KUKA KRL program: EPS_2_251626_SANMH03_A_20260107075954.src

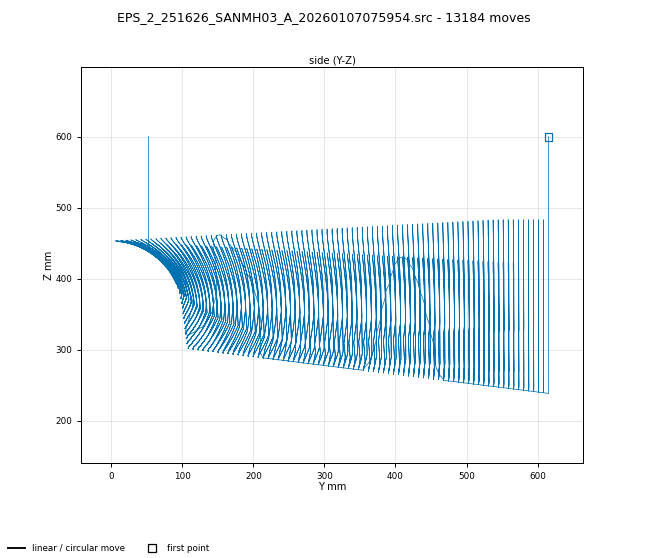
[picture p0: tool path of EPS_2_251626_SANMH03_A_20260107075954.src, 13184 of 13186 moves have a stored position in this frame; points joined in program order, loops and branches not executed]
&ACCESS RVP
&REL 4
&COMMENT QRS 19112012
&PARAM EDITMASK = *
DEF PART()
EXT BAS (BAS_COMMAND :IN,REAL :IN )
INT I
BAS (#INITMOV,0 )

;KUKA QRS Post kuka4.cps  Date:22-06-2017 !

File_ID=2961

QRS_PRE_INIT()

;Init var - Until changes are made in qrs_pre_init
Outlet_Square_prg=0
Inlet_1_Square_prg=0
Inlet_2_Square_prg=0
Inlet_3_Square_prg=0
Inlet_4_Square_prg=0
Inlet_5_Square_prg=0

Outlet_1={X 0.000, Y 541.230, Z 408.000, B 0.000, E1 0.000 }
Inlet_1={X 0.000, Y 545.490, Z 348.000, B 0.000, E1 180.000 }
Outlet_1_type=150
Inlet_1_type=150
;QRS#1=Sidecore dimensions
;QRS#2=150-6" PVC SDR 28
;QRS#3=150-6" PVC SDR 28
;QRS#4=
;QRS#5=
;QRS#6=
;QRS#7=
;QRS#8=
;QRS#9=10-06 PSX
;QRS#10=10-06 PSX
;QRS#11=
;QRS#12=
;QRS#13=
;QRS#14=
;QRS#15=
;QRS#16=1220x127x762 2,5'
;QRS#17=EPS Height
;QRS#18=483
;QRS#19=*
;QRS#20= UPDATED VERSION 22-06-2017
;QRS#21=*
Outlet_Square=070
Inlet_1_Square=070
Inlet_2_Square=0
Inlet_3_Square=0
Inlet_4_Square=0
Inlet_5_Square=0
Mill_Square=1
Outlet_Square_Prg=203
Inlet_1_Square_prg=203

QRS_INIT()

$ADVANCE=5

; T1
PTP {E1 173.651,E2 173.651}
PTP {X 0,Y 615.452,A -85,B 0,C 180,E1 173.651,E2 173.651,E3 0,E4 0,E5 0,E6 0}
QRS_SPEED_INIT()
LIN {X 0,Y 615.452,Z 600,A -85,B 0,C 180,E1 173.651,E2 173.651,E3 0,E4 0,E5 0,E6 0} C_VEL
LIN {X 0,Y 615.452,Z 248.689,A -85,B 0,C 180,E1 173.651,E2 173.651} C_VEL
LIN {X 0,Y 615.452,Z 240.511,A -85,B 0,C 180,E1 173.651,E2 173.651} C_VEL
LIN {X 0,Y 615.435,Z 238.511,A -85,B 0,C 180,E1 173.465,E2 173.465} C_VEL
LIN {X 0,Y 615.433,Z 238.511,A -85,B 0,C 180,E1 171.463,E2 171.463} C_VEL
LIN {X 0,Y 615.423,Z 238.51,A -85,B 0,C 180,E1 169.144,E2 169.144} C_VEL
LIN {X 0,Y 615.439,Z 238.509,A -85,B 0,C 180,E1 166.798,E2 166.798} C_VEL
LIN {X 0,Y 615.477,Z 238.513,A -85,B 0,C 180,E1 164.094,E2 164.094} C_VEL
LIN {X 0,Y 615.424,Z 238.51,A -85,B 0,C 180,E1 161.352,E2 161.352} C_VEL
LIN {X 0,Y 615.486,Z 238.507,A -85,B 0,C 180,E1 158.568,E2 158.568} C_VEL
LIN {X 0,Y 615.431,Z 238.51,A -85,B 0,C 180,E1 155.726,E2 155.726} C_VEL
LIN {X 0,Y 615.424,Z 238.51,A -85,B 0,C 180,E1 153.553,E2 153.553} C_VEL
LIN {X 0,Y 615.493,Z 238.51,A -85,B 0,C 180,E1 150.594,E2 150.594} C_VEL
LIN {X 0,Y 615.469,Z 238.512,A -85,B 0,C 180,E1 148.313,E2 148.313} C_VEL
LIN {X 0,Y 615.434,Z 238.51,A -85,B 0,C 180,E1 145.975,E2 145.975} C_VEL
LIN {X 0,Y 615.428,Z 238.509,A -85,B 0,C 180,E1 143.571,E2 143.571} C_VEL
LIN {X 0,Y 615.49,Z 238.506,A -85,B 0,C 180,E1 140.938,E2 140.938} C_VEL
LIN {X 0,Y 615.471,Z 238.512,A -85,B 0,C 180,E1 138.525,E2 138.525} C_VEL
LIN {X 0,Y 615.429,Z 238.509,A -85,B 0,C 180,E1 136.008,E2 136.008} C_VEL
LIN {X 0,Y 615.428,Z 238.509,A -85,B 0,C 180,E1 133.992,E2 133.992} C_VEL
LIN {X 0,Y 615.45,Z 238.507,A -85,B 0,C 180,E1 131.477,E2 131.477} C_VEL
LIN {X 0,Y 615.493,Z 238.513,A -85,B 0,C 180,E1 128.904,E2 128.904} C_VEL
LIN {X 0,Y 615.439,Z 238.51,A -85,B 0,C 180,E1 126.428,E2 126.428} C_VEL
LIN {X 0,Y 615.43,Z 238.508,A -85,B 0,C 180,E1 124.026,E2 124.026} C_VEL
LIN {X 0,Y 615.485,Z 238.516,A -85,B 0,C 180,E1 121.085,E2 121.085} C_VEL
LIN {X 0,Y 615.433,Z 238.509,A -85,B 0,C 180,E1 118.441,E2 118.441} C_VEL
LIN {X 0,Y 615.432,Z 238.509,A -85,B 0,C 180,E1 116.447,E2 116.447} C_VEL
LIN {X 0,Y 615.442,Z 238.507,A -85,B 0,C 180,E1 113.998,E2 113.998} C_VEL
LIN {X 0,Y 615.498,Z 238.508,A -85,B 0,C 180,E1 111.432,E2 111.432} C_VEL
LIN {X 0,Y 615.432,Z 238.509,A -85,B 0,C 180,E1 108.589,E2 108.589} C_VEL
LIN {X 0,Y 615.432,Z 238.508,A -85,B 0,C 180,E1 106.413,E2 106.413} C_VEL
LIN {X 0,Y 615.476,Z 238.722,A -85,B 0,C 180,E1 105.821,E2 105.821} C_VEL
LIN {X 0,Y 615.454,Z 250.521,A -85,B 0,C 180,E1 103.202,E2 103.202} C_VEL
LIN {X 0,Y 615.419,Z 261.215,A -85,B 0,C 180,E1 100.854,E2 100.854} C_VEL
LIN {X 0,Y 615.464,Z 264.873,A -85,B 0,C 180,E1 100.05,E2 100.05} C_VEL
LIN {X 0,Y 615.43,Z 339.723,A -85,B 0,C 180,E1 99.159,E2 99.159} C_VEL
LIN {X 0,Y 615.423,Z 347.907,A -85,B 0,C 180,E1 98.993,E2 98.993} C_VEL
LIN {X 0,Y 615.423,Z 356.463,A -85,B 0,C 180,E1 98.745,E2 98.745} C_VEL
LIN {X 0,Y 615.437,Z 364.07,A -85,B 0,C 180,E1 98.455,E2 98.455} C_VEL
LIN {X 0,Y 615.485,Z 372.58,A -85,B 0,C 180,E1 98.041,E2 98.041} C_VEL
LIN {X 0,Y 615.485,Z 380.745,A -85,B 0,C 180,E1 97.546,E2 97.546} C_VEL
LIN {X 0,Y 615.491,Z 387.386,A -85,B 0,C 180,E1 97.058,E2 97.058} C_VEL
LIN {X 0,Y 615.498,Z 393.181,A -85,B 0,C 180,E1 96.557,E2 96.557} C_VEL
LIN {X 0,Y 615.499,Z 399.532,A -85,B 0,C 180,E1 95.899,E2 95.899} C_VEL
LIN {X 0,Y 615.495,Z 405.982,A -85,B 0,C 180,E1 95.077,E2 95.077} C_VEL
LIN {X 0,Y 615.492,Z 411.121,A -85,B 0,C 180,E1 94.257,E2 94.257} C_VEL
LIN {X 0,Y 615.493,Z 415.885,A -85,B 0,C 180,E1 93.273,E2 93.273} C_VEL
LIN {X 0,Y 615.493,Z 418.199,A -85,B 0,C 180,E1 92.618,E2 92.618} C_VEL
LIN {X 0,Y 615.5,Z 419.975,A -85,B 0,C 180,E1 91.963,E2 91.963} C_VEL
LIN {X 0,Y 615.492,Z 421.266,A -85,B 0,C 180,E1 91.309,E2 91.309} C_VEL
LIN {X 0,Y 615.491,Z 422.083,A -85,B 0,C 180,E1 90.655,E2 90.655} C_VEL
LIN {X 0,Y 615.492,Z 422.384,A -85,B 0,C 180,E1 90,E2 90} C_VEL
LIN {X 0,Y 615.492,Z 422.125,A -85,B 0,C 180,E1 89.346,E2 89.346} C_VEL
LIN {X 0,Y 615.494,Z 421.394,A -85,B 0,C 180,E1 88.692,E2 88.692} C_VEL
LIN {X 0,Y 615.5,Z 420.195,A -85,B 0,C 180,E1 88.037,E2 88.037} C_VEL
LIN {X 0,Y 615.49,Z 417.377,A -85,B 0,C 180,E1 87.055,E2 87.055} C_VEL
LIN {X 0,Y 615.492,Z 414.811,A -85,B 0,C 180,E1 86.4,E2 86.4} C_VEL
LIN {X 0,Y 615.495,Z 409.745,A -85,B 0,C 180,E1 85.416,E2 85.416} C_VEL
LIN {X 0,Y 615.496,Z 404.29,A -85,B 0,C 180,E1 84.595,E2 84.595} C_VEL
LIN {X 0,Y 615.497,Z 397.456,A -85,B 0,C 180,E1 83.773,E2 83.773} C_VEL
LIN {X 0,Y 615.497,Z 390.421,A -85,B 0,C 180,E1 83.1,E2 83.1} C_VEL
LIN {X 0,Y 615.487,Z 382.077,A -85,B 0,C 180,E1 82.455,E2 82.455} C_VEL
LIN {X 0,Y 615.495,Z 374.202,A -85,B 0,C 180,E1 81.96,E2 81.96} C_VEL
LIN {X 0,Y 615.445,Z 366.093,A -85,B 0,C 180,E1 81.546,E2 81.546} C_VEL
LIN {X 0,Y 615.428,Z 357.89,A -85,B 0,C 180,E1 81.215,E2 81.215} C_VEL
LIN {X 0,Y 615.429,Z 349.874,A -85,B 0,C 180,E1 80.966,E2 80.966} C_VEL
LIN {X 0,Y 615.439,Z 340.208,A -85,B 0,C 180,E1 80.759,E2 80.759} C_VEL
LIN {X 0,Y 615.463,Z 264.814,A -85,B 0,C 180,E1 79.847,E2 79.847} C_VEL
LIN {X 0,Y 615.422,Z 253.988,A -85,B 0,C 180,E1 77.469,E2 77.469} C_VEL
LIN {X 0,Y 615.432,Z 243.324,A -85,B 0,C 180,E1 75.112,E2 75.112} C_VEL
LIN {X 0,Y 615.456,Z 238.508,A -85,B 0,C 180,E1 74.031,E2 74.031} C_VEL
LIN {X 0,Y 615.425,Z 238.51,A -85,B 0,C 180,E1 71.352,E2 71.352} C_VEL
LIN {X 0,Y 615.497,Z 238.511,A -85,B 0,C 180,E1 68.569,E2 68.569} C_VEL
LIN {X 0,Y 615.425,Z 238.509,A -85,B 0,C 180,E1 65.726,E2 65.726} C_VEL
LIN {X 0,Y 615.424,Z 238.51,A -85,B 0,C 180,E1 63.553,E2 63.553} C_VEL
LIN {X 0,Y 615.481,Z 238.51,A -85,B 0,C 180,E1 60.594,E2 60.594} C_VEL
LIN {X 0,Y 615.449,Z 238.508,A -85,B 0,C 180,E1 58.313,E2 58.313} C_VEL
LIN {X 0,Y 615.423,Z 238.51,A -85,B 0,C 180,E1 55.975,E2 55.975} C_VEL
LIN {X 0,Y 615.483,Z 238.512,A -85,B 0,C 180,E1 53.064,E2 53.064} C_VEL
LIN {X 0,Y 615.429,Z 238.51,A -85,B 0,C 180,E1 50.246,E2 50.246} C_VEL
LIN {X 0,Y 615.42,Z 238.511,A -85,B 0,C 180,E1 47.927,E2 47.927} C_VEL
LIN {X 0,Y 615.425,Z 238.511,A -85,B 0,C 180,E1 45.846,E2 45.846} C_VEL
LIN {X 0,Y 615.487,Z 238.512,A -85,B 0,C 180,E1 43.245,E2 43.245} C_VEL
LIN {X 0,Y 615.44,Z 238.509,A -85,B 0,C 180,E1 40.61,E2 40.61} C_VEL
LIN {X 0,Y 615.467,Z 238.509,A -85,B 0,C 180,E1 38.906,E2 38.906} C_VEL
LIN {X 0,Y 615.424,Z 238.51,A -85,B 0,C 180,E1 36.429,E2 36.429} C_VEL
LIN {X 0,Y 615.471,Z 238.513,A -85,B 0,C 180,E1 33.533,E2 33.533} C_VEL
LIN {X 0,Y 615.448,Z 238.509,A -85,B 0,C 180,E1 30.922,E2 30.922} C_VEL
LIN {X 0,Y 615.42,Z 238.51,A -85,B 0,C 180,E1 28.44,E2 28.44} C_VEL
LIN {X 0,Y 615.472,Z 238.512,A -85,B 0,C 180,E1 25.717,E2 25.717} C_VEL
LIN {X 0,Y 615.428,Z 238.51,A -85,B 0,C 180,E1 22.847,E2 22.847} C_VEL
LIN {X 0,Y 615.419,Z 238.511,A -85,B 0,C 180,E1 20.542,E2 20.542} C_VEL
LIN {X 0,Y 615.462,Z 238.512,A -85,B 0,C 180,E1 17.958,E2 17.958} C_VEL
LIN {X 0,Y 615.443,Z 238.51,A -85,B 0,C 180,E1 15.227,E2 15.227} C_VEL
LIN {X 0,Y 615.437,Z 238.51,A -85,B 0,C 180,E1 13.202,E2 13.202} C_VEL
LIN {X 0,Y 615.417,Z 238.511,A -85,B 0,C 180,E1 10.857,E2 10.857} C_VEL
LIN {X 0,Y 615.427,Z 238.511,A -85,B 0,C 180,E1 8.538,E2 8.538} C_VEL
LIN {X 0,Y 615.498,Z 238.511,A -85,B 0,C 180,E1 5.899,E2 5.899} C_VEL
LIN {X 0,Y 615.426,Z 238.511,A -85,B 0,C 180,E1 3.273,E2 3.273} C_VEL
LIN {X 0,Y 615.425,Z 238.511,A -85,B 0,C 180,E1 1.309,E2 1.309} C_VEL
LIN {X 0,Y 615.425,Z 238.511,A -85,B 0,C 180,E1 -0.654,E2 -0.654} C_VEL
LIN {X 0,Y 615.424,Z 238.511,A -85,B 0,C 180,E1 -2.618,E2 -2.618} C_VEL
LIN {X 0,Y 615.424,Z 238.511,A -85,B 0,C 180,E1 -4.585,E2 -4.585} C_VEL
LIN {X 0,Y 615.423,Z 238.511,A -85,B 0,C 180,E1 -6.557,E2 -6.557} C_VEL
LIN {X 0,Y 615.422,Z 238.511,A -85,B 0,C 180,E1 -8.537,E2 -8.537} C_VEL
LIN {X 0,Y 615.417,Z 238.512,A -85,B 0,C 180,E1 -10.857,E2 -10.857} C_VEL
LIN {X 0,Y 615.441,Z 238.512,A -85,B 0,C 180,E1 -13.202,E2 -13.202} C_VEL
LIN {X 0,Y 615.461,Z 238.511,A -85,B 0,C 180,E1 -15.906,E2 -15.906} C_VEL
LIN {X 0,Y 615.415,Z 238.512,A -85,B 0,C 180,E1 -18.648,E2 -18.648} C_VEL
LIN {X 0,Y 615.493,Z 238.512,A -85,B 0,C 180,E1 -21.432,E2 -21.432} C_VEL
LIN {X 0,Y 615.417,Z 238.511,A -85,B 0,C 180,E1 -24.275,E2 -24.275} C_VEL
LIN {X 0,Y 615.415,Z 238.512,A -85,B 0,C 180,E1 -26.447,E2 -26.447} C_VEL
LIN {X 0,Y 615.478,Z 238.514,A -85,B 0,C 180,E1 -29.407,E2 -29.407} C_VEL
LIN {X 0,Y 615.445,Z 238.511,A -85,B 0,C 180,E1 -31.688,E2 -31.688} C_VEL
LIN {X 0,Y 615.418,Z 238.512,A -85,B 0,C 180,E1 -34.026,E2 -34.026} C_VEL
LIN {X 0,Y 615.464,Z 238.513,A -85,B 0,C 180,E1 -36.935,E2 -36.935} C_VEL
LIN {X 0,Y 615.422,Z 238.512,A -85,B 0,C 180,E1 -39.755,E2 -39.755} C_VEL
LIN {X 0,Y 615.413,Z 238.512,A -85,B 0,C 180,E1 -42.073,E2 -42.073} C_VEL
LIN {X 0,Y 615.415,Z 238.512,A -85,B 0,C 180,E1 -44.156,E2 -44.156} C_VEL
LIN {X 0,Y 615.471,Z 238.512,A -85,B 0,C 180,E1 -46.755,E2 -46.755} C_VEL
LIN {X 0,Y 615.435,Z 238.512,A -85,B 0,C 180,E1 -49.39,E2 -49.39} C_VEL
LIN {X 0,Y 615.465,Z 238.512,A -85,B 0,C 180,E1 -51.095,E2 -51.095} C_VEL
LIN {X 0,Y 615.417,Z 238.512,A -85,B 0,C 180,E1 -53.571,E2 -53.571} C_VEL
LIN {X 0,Y 615.46,Z 238.512,A -85,B 0,C 180,E1 -56.47,E2 -56.47} C_VEL
LIN {X 0,Y 615.444,Z 238.512,A -85,B 0,C 180,E1 -59.078,E2 -59.078} C_VEL
LIN {X 0,Y 615.412,Z 238.512,A -85,B 0,C 180,E1 -61.563,E2 -61.563} C_VEL
LIN {X 0,Y 615.409,Z 238.513,A -85,B 0,C 180,E1 -63.553,E2 -63.553} C_VEL
LIN {X 0,Y 615.431,Z 238.512,A -85,B 0,C 180,E1 -66.003,E2 -66.003} C_VEL
LIN {X 0,Y 615.422,Z 238.609,A -85,B 0,C 180,E1 -67.838,E2 -67.838} C_VEL
LIN {X 0,Y 615.475,Z 257.737,A -85,B 0,C 180,E1 -70.662,E2 -70.662} C_VEL
LIN {X 0,Y 615.482,Z 276.679,A -85,B 0,C 180,E1 -73.414,E2 -73.414} C_VEL
LIN {X 0,Y 615.488,Z 296.786,A -85,B 0,C 180,E1 -76.295,E2 -76.295} C_VEL
LIN {X 0,Y 615.448,Z 316.82,A -85,B 0,C 180,E1 -79.131,E2 -79.131} C_VEL
LIN {X 0,Y 615.46,Z 322.04,A -85,B 0,C 180,E1 -79.868,E2 -79.868} C_VEL
LIN {X 0,Y 615.446,Z 399.981,A -85,B 0,C 180,E1 -80.801,E2 -80.801} C_VEL
LIN {X 0,Y 615.436,Z 409.728,A -85,B 0,C 180,E1 -81.008,E2 -81.008} C_VEL
LIN {X 0,Y 615.436,Z 420.18,A -85,B 0,C 180,E1 -81.339,E2 -81.339} C_VEL
LIN {X 0,Y 615.471,Z 430.44,A -85,B 0,C 180,E1 -81.794,E2 -81.794} C_VEL
LIN {X 0,Y 615.489,Z 440.204,A -85,B 0,C 180,E1 -82.372,E2 -82.372} C_VEL
LIN {X 0,Y 615.494,Z 447.938,A -85,B 0,C 180,E1 -82.942,E2 -82.942} C_VEL
LIN {X 0,Y 615.497,Z 455.338,A -85,B 0,C 180,E1 -83.608,E2 -83.608} C_VEL
LIN {X 0,Y 615.498,Z 462.74,A -85,B 0,C 180,E1 -84.431,E2 -84.431} C_VEL
LIN {X 0,Y 615.497,Z 468.535,A -85,B 0,C 180,E1 -85.252,E2 -85.252} C_VEL
LIN {X 0,Y 615.496,Z 473.102,A -85,B 0,C 180,E1 -86.072,E2 -86.072} C_VEL
LIN {X 0,Y 615.492,Z 476.07,A -85,B 0,C 180,E1 -86.727,E2 -86.727} C_VEL
LIN {X 0,Y 615.494,Z 478.358,A -85,B 0,C 180,E1 -87.383,E2 -87.383} C_VEL
LIN {X 0,Y 615.5,Z 480.086,A -85,B 0,C 180,E1 -88.037,E2 -88.037} C_VEL
LIN {X 0,Y 615.493,Z 481.33,A -85,B 0,C 180,E1 -88.692,E2 -88.692} C_VEL
LIN {X 0,Y 615.492,Z 482.104,A -85,B 0,C 180,E1 -89.346,E2 -89.346} C_VEL
LIN {X 0,Y 615.491,Z 482.389,A -85,B 0,C 180,E1 -90,E2 -90} C_VEL
LIN {X 0,Y 615.491,Z 482.104,A -85,B 0,C 180,E1 -90.655,E2 -90.655} C_VEL
LIN {X 0,Y 615.493,Z 481.329,A -85,B 0,C 180,E1 -91.309,E2 -91.309} C_VEL
LIN {X 0,Y 615.5,Z 480.084,A -85,B 0,C 180,E1 -91.963,E2 -91.963} C_VEL
LIN {X 0,Y 615.488,Z 477.22,A -85,B 0,C 180,E1 -92.946,E2 -92.946} C_VEL
LIN {X 0,Y 615.491,Z 474.602,A -85,B 0,C 180,E1 -93.601,E2 -93.601} C_VEL
LIN {X 0,Y 615.495,Z 469.48,A -85,B 0,C 180,E1 -94.585,E2 -94.585} C_VEL
LIN {X 0,Y 615.495,Z 463.966,A -85,B 0,C 180,E1 -95.406,E2 -95.406} C_VEL
LIN {X 0,Y 615.498,Z 457.015,A -85,B 0,C 180,E1 -96.228,E2 -96.228} C_VEL
LIN {X 0,Y 615.496,Z 449.857,A -85,B 0,C 180,E1 -96.901,E2 -96.901} C_VEL
LIN {X 0,Y 615.485,Z 442.618,A -85,B 0,C 180,E1 -97.463,E2 -97.463} C_VEL
LIN {X 0,Y 615.495,Z 434.863,A -85,B 0,C 180,E1 -97.958,E2 -97.958} C_VEL
LIN {X 0,Y 615.454,Z 426.917,A -85,B 0,C 180,E1 -98.372,E2 -98.372} C_VEL
LIN {X 0,Y 615.434,Z 417.763,A -85,B 0,C 180,E1 -98.744,E2 -98.744} C_VEL
LIN {X 0,Y 615.436,Z 409.701,A -85,B 0,C 180,E1 -98.993,E2 -98.993} C_VEL
LIN {X 0,Y 615.446,Z 399.938,A -85,B 0,C 180,E1 -99.2,E2 -99.2} C_VEL
LIN {X 0,Y 615.46,Z 322.035,A -85,B 0,C 180,E1 -100.133,E2 -100.133} C_VEL
LIN {X 0,Y 615.468,Z 303.881,A -85,B 0,C 180,E1 -102.698,E2 -102.698} C_VEL
LIN {X 0,Y 615.486,Z 283.774,A -85,B 0,C 180,E1 -105.566,E2 -105.566} C_VEL
LIN {X 0,Y 615.469,Z 263.911,A -85,B 0,C 180,E1 -108.437,E2 -108.437} C_VEL
LIN {X 0,Y 615.439,Z 247.065,A -85,B 0,C 180,E1 -110.908,E2 -110.908} C_VEL
LIN {X 0,Y 615.42,Z 238.512,A -85,B 0,C 180,E1 -112.187,E2 -112.187} C_VEL
LIN {X 0,Y 615.414,Z 238.512,A -85,B 0,C 180,E1 -114.275,E2 -114.275} C_VEL
LIN {X 0,Y 615.41,Z 238.513,A -85,B 0,C 180,E1 -116.448,E2 -116.448} C_VEL
LIN {X 0,Y 615.478,Z 238.516,A -85,B 0,C 180,E1 -119.407,E2 -119.407} C_VEL
LIN {X 0,Y 615.446,Z 238.512,A -85,B 0,C 180,E1 -121.688,E2 -121.688} C_VEL
LIN {X 0,Y 615.417,Z 238.512,A -85,B 0,C 180,E1 -124.027,E2 -124.027} C_VEL
LIN {X 0,Y 615.463,Z 238.512,A -85,B 0,C 180,E1 -126.934,E2 -126.934} C_VEL
LIN {X 0,Y 615.426,Z 238.512,A -85,B 0,C 180,E1 -129.755,E2 -129.755} C_VEL
LIN {X 0,Y 615.414,Z 238.512,A -85,B 0,C 180,E1 -132.073,E2 -132.073} C_VEL
LIN {X 0,Y 615.415,Z 238.512,A -85,B 0,C 180,E1 -134.156,E2 -134.156} C_VEL
LIN {X 0,Y 615.414,Z 238.512,A -85,B 0,C 180,E1 -136.01,E2 -136.01} C_VEL
LIN {X 0,Y 615.445,Z 238.511,A -85,B 0,C 180,E1 -138.523,E2 -138.523} C_VEL
LIN {X 0,Y 615.472,Z 238.512,A -85,B 0,C 180,E1 -141.095,E2 -141.095} C_VEL
LIN {X 0,Y 615.422,Z 238.512,A -85,B 0,C 180,E1 -143.571,E2 -143.571} C_VEL
LIN {X 0,Y 615.418,Z 238.511,A -85,B 0,C 180,E1 -145.974,E2 -145.974} C_VEL
LIN {X 0,Y 615.443,Z 238.511,A -85,B 0,C 180,E1 -148.312,E2 -148.312} C_VEL
LIN {X 0,Y 615.478,Z 238.513,A -85,B 0,C 180,E1 -150.593,E2 -150.593} C_VEL
LIN {X 0,Y 615.418,Z 238.511,A -85,B 0,C 180,E1 -153.553,E2 -153.553} C_VEL
LIN {X 0,Y 615.433,Z 238.511,A -85,B 0,C 180,E1 -156.003,E2 -156.003} C_VEL
LIN {X 0,Y 615.498,Z 238.513,A -85,B 0,C 180,E1 -158.569,E2 -158.569} C_VEL
LIN {X 0,Y 615.418,Z 238.511,A -85,B 0,C 180,E1 -161.415,E2 -161.415} C_VEL
LIN {X 0,Y 615.462,Z 238.51,A -85,B 0,C 180,E1 -164.094,E2 -164.094} C_VEL
LIN {X 0,Y 615.445,Z 238.512,A -85,B 0,C 180,E1 -166.798,E2 -166.798} C_VEL
LIN {X 0,Y 615.421,Z 238.511,A -85,B 0,C 180,E1 -169.144,E2 -169.144} C_VEL
LIN {X 0,Y 615.424,Z 238.51,A -85,B 0,C 180,E1 -171.463,E2 -171.463} C_VEL
LIN {X 0,Y 615.496,Z 238.508,A -85,B 0,C 180,E1 -174.102,E2 -174.102} C_VEL
LIN {X 0,Y 615.435,Z 238.511,A -85,B 0,C 180,E1 -176.727,E2 -176.727} C_VEL
LIN {X 0,Y 615.435,Z 238.511,A -85,B 0,C 180,E1 -178.691,E2 -178.691} C_VEL
LIN {X 0,Y 615.434,Z 238.511,A -85,B 0,C 180,E1 -180.654,E2 -180.654} C_VEL
LIN {X 0,Y 615.435,Z 238.511,A -85,B 0,C 180,E1 -182.618,E2 -182.618} C_VEL
LIN {X 0,Y 615.434,Z 238.511,A -85,B 0,C 180,E1 -184.585,E2 -184.585} C_VEL
LIN {X 0,Y 615.435,Z 238.511,A -85,B 0,C 180,E1 -186.535,E2 -186.535} C_VEL
LIN {X 0,Y 614.753,Z 238.655,A -85,B 0,C 180,E1 -187.081,E2 -187.081} C_VEL
LIN {X 0,Y 611.913,Z 239.08,A -85,B 0,C 180,E1 -187.967,E2 -187.967} C_VEL
LIN {X 0,Y 609.529,Z 239.382,A -85,B 0,C 180,E1 -188.68,E2 -188.68} C_VEL
LIN {X 0,Y 608.51,Z 239.496,A -85,B 0,C 180,E1 -189.23,E2 -189.23} C_VEL
LIN {X 0,Y 608.429,Z 239.505,A -85,B 0,C 180,E1 -189.416,E2 -189.416} C_VEL
LIN {X 0,Y 608.449,Z 239.509,A -85,B 0,C 180,E1 -192,E2 -192} C_VEL
LIN {X 0,Y 608.396,Z 239.507,A -85,B 0,C 180,E1 -194.723,E2 -194.723} C_VEL
LIN {X 0,Y 608.428,Z 239.509,A -85,B 0,C 180,E1 -197.477,E2 -197.477} C_VEL
LIN {X 0,Y 608.42,Z 239.506,A -85,B 0,C 180,E1 -200.276,E2 -200.276} C_VEL
LIN {X 0,Y 608.397,Z 239.507,A -85,B 0,C 180,E1 -202.462,E2 -202.462} C_VEL
LIN {X 0,Y 608.412,Z 239.505,A -85,B 0,C 180,E1 -204.573,E2 -204.573} C_VEL
LIN {X 0,Y 608.46,Z 239.504,A -85,B 0,C 180,E1 -207.204,E2 -207.204} C_VEL
LIN {X 0,Y 608.419,Z 239.507,A -85,B 0,C 180,E1 -209.963,E2 -209.963} C_VEL
LIN {X 0,Y 608.412,Z 239.505,A -85,B 0,C 180,E1 -212.515,E2 -212.515} C_VEL
LIN {X 0,Y 608.417,Z 239.507,A -85,B 0,C 180,E1 -214.901,E2 -214.901} C_VEL
LIN {X 0,Y 608.438,Z 239.506,A -85,B 0,C 180,E1 -217.749,E2 -217.749} C_VEL
LIN {X 0,Y 608.403,Z 239.506,A -85,B 0,C 180,E1 -220.323,E2 -220.323} C_VEL
LIN {X 0,Y 608.447,Z 239.507,A -85,B 0,C 180,E1 -222.96,E2 -222.96} C_VEL
LIN {X 0,Y 608.414,Z 239.507,A -85,B 0,C 180,E1 -225.74,E2 -225.74} C_VEL
LIN {X 0,Y 608.413,Z 239.505,A -85,B 0,C 180,E1 -227.934,E2 -227.934} C_VEL
LIN {X 0,Y 608.438,Z 239.506,A -85,B 0,C 180,E1 -230.706,E2 -230.706} C_VEL
LIN {X 0,Y 608.454,Z 239.51,A -85,B 0,C 180,E1 -233.085,E2 -233.085} C_VEL
LIN {X 0,Y 608.437,Z 239.504,A -85,B 0,C 180,E1 -235.528,E2 -235.528} C_VEL
LIN {X 0,Y 608.422,Z 239.504,A -85,B 0,C 180,E1 -237.903,E2 -237.903} C_VEL
LIN {X 0,Y 608.433,Z 239.504,A -85,B 0,C 180,E1 -240.218,E2 -240.218} C_VEL
LIN {X 0,Y 608.48,Z 239.507,A -85,B 0,C 180,E1 -242.793,E2 -242.793} C_VEL
LIN {X 0,Y 608.421,Z 239.505,A -85,B 0,C 180,E1 -245.427,E2 -245.427} C_VEL
LIN {X 0,Y 608.458,Z 239.503,A -85,B 0,C 180,E1 -248.308,E2 -248.308} C_VEL
LIN {X 0,Y 608.418,Z 239.506,A -85,B 0,C 180,E1 -251.299,E2 -251.299} C_VEL
LIN {X 0,Y 608.455,Z 239.58,A -85,B 0,C 180,E1 -254.142,E2 -254.142} C_VEL
LIN {X 0,Y 608.411,Z 252.299,A -85,B 0,C 180,E1 -256.982,E2 -256.982} C_VEL
LIN {X 0,Y 608.401,Z 264.922,A -85,B 0,C 180,E1 -259.769,E2 -259.769} C_VEL
LIN {X 0,Y 608.426,Z 265.209,A -85,B 0,C 180,E1 -259.833,E2 -259.833} C_VEL
LIN {X 0,Y 608.458,Z 340.233,A -85,B 0,C 180,E1 -260.736,E2 -260.736} C_VEL
LIN {X 0,Y 608.448,Z 349.939,A -85,B 0,C 180,E1 -260.945,E2 -260.945} C_VEL
LIN {X 0,Y 608.433,Z 361.53,A -85,B 0,C 180,E1 -261.321,E2 -261.321} C_VEL
LIN {X 0,Y 608.462,Z 371.427,A -85,B 0,C 180,E1 -261.782,E2 -261.782} C_VEL
LIN {X 0,Y 608.468,Z 379.881,A -85,B 0,C 180,E1 -262.283,E2 -262.283} C_VEL
LIN {X 0,Y 608.459,Z 387.85,A -85,B 0,C 180,E1 -262.867,E2 -262.867} C_VEL
LIN {X 0,Y 608.468,Z 394.901,A -85,B 0,C 180,E1 -263.496,E2 -263.496} C_VEL
LIN {X 0,Y 608.458,Z 401.393,A -85,B 0,C 180,E1 -264.199,E2 -264.199} C_VEL
LIN {X 0,Y 608.437,Z 407.639,A -85,B 0,C 180,E1 -265.03,E2 -265.03} C_VEL
LIN {X 0,Y 608.434,Z 413.423,A -85,B 0,C 180,E1 -266.026,E2 -266.026} C_VEL
LIN {X 0,Y 608.447,Z 417.629,A -85,B 0,C 180,E1 -267.02,E2 -267.02} C_VEL
LIN {X 0,Y 608.444,Z 420.569,A -85,B 0,C 180,E1 -268.014,E2 -268.014} C_VEL
LIN {X 0,Y 608.445,Z 421.869,A -85,B 0,C 180,E1 -268.676,E2 -268.676} C_VEL
LIN {X 0,Y 608.434,Z 422.692,A -85,B 0,C 180,E1 -269.338,E2 -269.338} C_VEL
LIN {X 0,Y 608.432,Z 422.995,A -85,B 0,C 180,E1 -270,E2 -270} C_VEL
LIN {X 0,Y 608.435,Z 422.735,A -85,B 0,C 180,E1 -270.661,E2 -270.661} C_VEL
LIN {X 0,Y 608.446,Z 421.998,A -85,B 0,C 180,E1 -271.323,E2 -271.323} C_VEL
LIN {X 0,Y 608.444,Z 420.788,A -85,B 0,C 180,E1 -271.985,E2 -271.985} C_VEL
LIN {X 0,Y 608.445,Z 417.943,A -85,B 0,C 180,E1 -272.979,E2 -272.979} C_VEL
LIN {X 0,Y 608.446,Z 415.353,A -85,B 0,C 180,E1 -273.642,E2 -273.642} C_VEL
LIN {X 0,Y 608.445,Z 410.247,A -85,B 0,C 180,E1 -274.637,E2 -274.637} C_VEL
LIN {X 0,Y 608.461,Z 404.751,A -85,B 0,C 180,E1 -275.468,E2 -275.468} C_VEL
LIN {X 0,Y 608.454,Z 397.149,A -85,B 0,C 180,E1 -276.374,E2 -276.374} C_VEL
LIN {X 0,Y 608.463,Z 388.952,A -85,B 0,C 180,E1 -277.132,E2 -277.132} C_VEL
LIN {X 0,Y 608.469,Z 381.204,A -85,B 0,C 180,E1 -277.716,E2 -277.716} C_VEL
LIN {X 0,Y 608.47,Z 373.04,A -85,B 0,C 180,E1 -278.217,E2 -278.217} C_VEL
LIN {X 0,Y 608.434,Z 364.54,A -85,B 0,C 180,E1 -278.636,E2 -278.636} C_VEL
LIN {X 0,Y 608.422,Z 353.345,A -85,B 0,C 180,E1 -279.055,E2 -279.055} C_VEL
LIN {X 0,Y 608.461,Z 341.959,A -85,B 0,C 180,E1 -279.327,E2 -279.327} C_VEL
LIN {X 0,Y 608.469,Z 321.042,A -85,B 0,C 180,E1 -279.599,E2 -279.599} C_VEL
LIN {X 0,Y 608.41,Z 265.143,A -85,B 0,C 180,E1 -280.272,E2 -280.272} C_VEL
LIN {X 0,Y 608.402,Z 252.707,A -85,B 0,C 180,E1 -283.017,E2 -283.017} C_VEL
LIN {X 0,Y 608.449,Z 240.462,A -85,B 0,C 180,E1 -285.75,E2 -285.75} C_VEL
LIN {X 0,Y 608.44,Z 239.504,A -85,B 0,C 180,E1 -286.008,E2 -286.008} C_VEL
LIN {X 0,Y 608.43,Z 239.505,A -85,B 0,C 180,E1 -288.87,E2 -288.87} C_VEL
LIN {X 0,Y 608.456,Z 239.505,A -85,B 0,C 180,E1 -291.692,E2 -291.692} C_VEL
LIN {X 0,Y 608.414,Z 239.506,A -85,B 0,C 180,E1 -294.572,E2 -294.572} C_VEL
LIN {X 0,Y 608.471,Z 239.508,A -85,B 0,C 180,E1 -297.206,E2 -297.206} C_VEL
LIN {X 0,Y 608.406,Z 239.506,A -85,B 0,C 180,E1 -299.961,E2 -299.961} C_VEL
LIN {X 0,Y 608.413,Z 239.506,A -85,B 0,C 180,E1 -302.515,E2 -302.515} C_VEL
LIN {X 0,Y 608.421,Z 239.511,A -85,B 0,C 180,E1 -304.901,E2 -304.901} C_VEL
LIN {X 0,Y 608.429,Z 239.504,A -85,B 0,C 180,E1 -307.749,E2 -307.749} C_VEL
LIN {X 0,Y 608.398,Z 239.508,A -85,B 0,C 180,E1 -310.323,E2 -310.323} C_VEL
LIN {X 0,Y 608.447,Z 239.511,A -85,B 0,C 180,E1 -312.96,E2 -312.96} C_VEL
LIN {X 0,Y 608.404,Z 239.506,A -85,B 0,C 180,E1 -315.74,E2 -315.74} C_VEL
LIN {X 0,Y 608.406,Z 239.506,A -85,B 0,C 180,E1 -317.934,E2 -317.934} C_VEL
LIN {X 0,Y 608.434,Z 239.512,A -85,B 0,C 180,E1 -320.706,E2 -320.706} C_VEL
LIN {X 0,Y 608.433,Z 239.507,A -85,B 0,C 180,E1 -323.083,E2 -323.083} C_VEL
LIN {X 0,Y 608.42,Z 239.504,A -85,B 0,C 180,E1 -325.527,E2 -325.527} C_VEL
LIN {X 0,Y 608.418,Z 239.505,A -85,B 0,C 180,E1 -327.903,E2 -327.903} C_VEL
LIN {X 0,Y 608.438,Z 239.507,A -85,B 0,C 180,E1 -330.219,E2 -330.219} C_VEL
LIN {X 0,Y 608.398,Z 239.508,A -85,B 0,C 180,E1 -333.223,E2 -333.223} C_VEL
LIN {X 0,Y 608.407,Z 239.506,A -85,B 0,C 180,E1 -335.427,E2 -335.427} C_VEL
LIN {X 0,Y 608.45,Z 239.51,A -85,B 0,C 180,E1 -338.308,E2 -338.308} C_VEL
LIN {X 0,Y 608.406,Z 239.506,A -85,B 0,C 180,E1 -341.3,E2 -341.3} C_VEL
LIN {X 0,Y 608.428,Z 239.508,A -85,B 0,C 180,E1 -343.905,E2 -343.905} C_VEL
LIN {X 0,Y 608.428,Z 239.507,A -85,B 0,C 180,E1 -346.643,E2 -346.643} C_VEL
LIN {X 0,Y 608.402,Z 239.507,A -85,B 0,C 180,E1 -349.349,E2 -349.349} C_VEL
LIN {X 0,Y 608.465,Z 239.508,A -85,B 0,C 180,E1 -352.033,E2 -352.033} C_VEL
LIN {X 0,Y 608.413,Z 239.506,A -85,B 0,C 180,E1 -354.698,E2 -354.698} C_VEL
LIN {X 0,Y 608.424,Z 239.505,A -85,B 0,C 180,E1 -357.352,E2 -357.352} C_VEL
LIN {X 0,Y 608.47,Z 239.507,A -85,B 0,C 180,E1 -360,E2 -360} C_VEL
LIN {X 0,Y 608.42,Z 239.505,A -85,B 0,C 180,E1 -362.648,E2 -362.648} C_VEL
LIN {X 0,Y 608.419,Z 239.507,A -85,B 0,C 180,E1 -365.302,E2 -365.302} C_VEL
LIN {X 0,Y 608.463,Z 239.506,A -85,B 0,C 180,E1 -367.967,E2 -367.967} C_VEL
LIN {X 0,Y 608.4,Z 239.507,A -85,B 0,C 180,E1 -370.651,E2 -370.651} C_VEL
LIN {X 0,Y 608.428,Z 239.509,A -85,B 0,C 180,E1 -373.357,E2 -373.357} C_VEL
LIN {X 0,Y 608.422,Z 239.507,A -85,B 0,C 180,E1 -376.095,E2 -376.095} C_VEL
LIN {X 0,Y 608.422,Z 239.505,A -85,B 0,C 180,E1 -378.871,E2 -378.871} C_VEL
LIN {X 0,Y 608.451,Z 239.507,A -85,B 0,C 180,E1 -381.692,E2 -381.692} C_VEL
LIN {X 0,Y 608.404,Z 239.506,A -85,B 0,C 180,E1 -384.573,E2 -384.573} C_VEL
LIN {X 0,Y 608.459,Z 239.507,A -85,B 0,C 180,E1 -387.205,E2 -387.205} C_VEL
LIN {X 0,Y 608.401,Z 239.508,A -85,B 0,C 180,E1 -389.962,E2 -389.962} C_VEL
LIN {X 0,Y 608.404,Z 239.507,A -85,B 0,C 180,E1 -392.515,E2 -392.515} C_VEL
LIN {X 0,Y 608.412,Z 239.511,A -85,B 0,C 180,E1 -394.901,E2 -394.901} C_VEL
LIN {X 0,Y 608.423,Z 239.505,A -85,B 0,C 180,E1 -397.75,E2 -397.75} C_VEL
LIN {X 0,Y 608.396,Z 239.508,A -85,B 0,C 180,E1 -400.324,E2 -400.324} C_VEL
LIN {X 0,Y 608.437,Z 239.512,A -85,B 0,C 180,E1 -402.961,E2 -402.961} C_VEL
LIN {X 0,Y 608.398,Z 239.507,A -85,B 0,C 180,E1 -405.742,E2 -405.742} C_VEL
LIN {X 0,Y 608.398,Z 239.507,A -85,B 0,C 180,E1 -407.934,E2 -407.934} C_VEL
LIN {X 0,Y 608.43,Z 239.511,A -85,B 0,C 180,E1 -410.707,E2 -410.707} C_VEL
LIN {X 0,Y 608.431,Z 239.508,A -85,B 0,C 180,E1 -413.084,E2 -413.084} C_VEL
LIN {X 0,Y 608.416,Z 239.505,A -85,B 0,C 180,E1 -415.528,E2 -415.528} C_VEL
LIN {X 0,Y 608.409,Z 239.506,A -85,B 0,C 180,E1 -417.903,E2 -417.903} C_VEL
LIN {X 0,Y 608.425,Z 239.507,A -85,B 0,C 180,E1 -420.219,E2 -420.219} C_VEL
LIN {X 0,Y 608.456,Z 239.507,A -85,B 0,C 180,E1 -422.797,E2 -422.797} C_VEL
LIN {X 0,Y 608.401,Z 239.507,A -85,B 0,C 180,E1 -425.427,E2 -425.427} C_VEL
LIN {X 0,Y 608.423,Z 239.662,A -85,B 0,C 180,E1 -427.727,E2 -427.727} C_VEL
LIN {X 0,Y 608.49,Z 251.996,A -85,B 0,C 180,E1 -429.576,E2 -429.576} C_VEL
LIN {X 0,Y 608.507,Z 270.816,A -85,B 0,C 180,E1 -432.352,E2 -432.352} C_VEL
LIN {X 0,Y 608.482,Z 289.806,A -85,B 0,C 180,E1 -435.109,E2 -435.109} C_VEL
LIN {X 0,Y 608.453,Z 308.795,A -85,B 0,C 180,E1 -437.831,E2 -437.831} C_VEL
LIN {X 0,Y 608.436,Z 322.296,A -85,B 0,C 180,E1 -439.75,E2 -439.75} C_VEL
LIN {X 0,Y 608.473,Z 400.467,A -85,B 0,C 180,E1 -440.695,E2 -440.695} C_VEL
LIN {X 0,Y 608.437,Z 410.09,A -85,B 0,C 180,E1 -440.904,E2 -440.904} C_VEL
LIN {X 0,Y 608.426,Z 421.627,A -85,B 0,C 180,E1 -441.28,E2 -441.28} C_VEL
LIN {X 0,Y 608.47,Z 432.239,A -85,B 0,C 180,E1 -441.783,E2 -441.783} C_VEL
LIN {X 0,Y 608.468,Z 440.547,A -85,B 0,C 180,E1 -442.284,E2 -442.284} C_VEL
LIN {X 0,Y 608.46,Z 448.405,A -85,B 0,C 180,E1 -442.868,E2 -442.868} C_VEL
LIN {X 0,Y 608.466,Z 455.359,A -85,B 0,C 180,E1 -443.496,E2 -443.496} C_VEL
LIN {X 0,Y 608.47,Z 463.194,A -85,B 0,C 180,E1 -444.366,E2 -444.366} C_VEL
LIN {X 0,Y 608.448,Z 469.029,A -85,B 0,C 180,E1 -445.197,E2 -445.197} C_VEL
LIN {X 0,Y 608.434,Z 473.632,A -85,B 0,C 180,E1 -446.026,E2 -446.026} C_VEL
LIN {X 0,Y 608.424,Z 476.623,A -85,B 0,C 180,E1 -446.689,E2 -446.689} C_VEL
LIN {X 0,Y 608.423,Z 478.932,A -85,B 0,C 180,E1 -447.352,E2 -447.352} C_VEL
LIN {X 0,Y 608.444,Z 480.679,A -85,B 0,C 180,E1 -448.015,E2 -448.015} C_VEL
LIN {X 0,Y 608.445,Z 481.934,A -85,B 0,C 180,E1 -448.677,E2 -448.677} C_VEL
LIN {X 0,Y 608.434,Z 482.714,A -85,B 0,C 180,E1 -449.339,E2 -449.339} C_VEL
LIN {X 0,Y 608.431,Z 483,A -85,B 0,C 180,E1 -450,E2 -450} C_VEL
LIN {X 0,Y 608.434,Z 482.713,A -85,B 0,C 180,E1 -450.662,E2 -450.662} C_VEL
LIN {X 0,Y 608.446,Z 481.933,A -85,B 0,C 180,E1 -451.324,E2 -451.324} C_VEL
LIN {X 0,Y 608.444,Z 480.677,A -85,B 0,C 180,E1 -451.986,E2 -451.986} C_VEL
LIN {X 0,Y 608.444,Z 477.785,A -85,B 0,C 180,E1 -452.98,E2 -452.98} C_VEL
LIN {X 0,Y 608.445,Z 475.145,A -85,B 0,C 180,E1 -453.643,E2 -453.643} C_VEL
LIN {X 0,Y 608.431,Z 469.983,A -85,B 0,C 180,E1 -454.638,E2 -454.638} C_VEL
LIN {X 0,Y 608.46,Z 464.427,A -85,B 0,C 180,E1 -455.468,E2 -455.468} C_VEL
LIN {X 0,Y 608.455,Z 456.67,A -85,B 0,C 180,E1 -456.376,E2 -456.376} C_VEL
LIN {X 0,Y 608.453,Z 449.411,A -85,B 0,C 180,E1 -457.05,E2 -457.05} C_VEL
LIN {X 0,Y 608.468,Z 441.755,A -85,B 0,C 180,E1 -457.633,E2 -457.633} C_VEL
LIN {X 0,Y 608.48,Z 433.714,A -85,B 0,C 180,E1 -458.134,E2 -458.134} C_VEL
LIN {X 0,Y 608.45,Z 425.382,A -85,B 0,C 180,E1 -458.553,E2 -458.553} C_VEL
LIN {X 0,Y 608.431,Z 416.879,A -85,B 0,C 180,E1 -458.888,E2 -458.888} C_VEL
LIN {X 0,Y 608.438,Z 407.572,A -85,B 0,C 180,E1 -459.16,E2 -459.16} C_VEL
LIN {X 0,Y 608.481,Z 396.528,A -85,B 0,C 180,E1 -459.369,E2 -459.369} C_VEL
LIN {X 0,Y 608.436,Z 322.291,A -85,B 0,C 180,E1 -460.251,E2 -460.251} C_VEL
LIN {X 0,Y 608.485,Z 302.856,A -85,B 0,C 180,E1 -463.016,E2 -463.016} C_VEL
LIN {X 0,Y 608.493,Z 282.68,A -85,B 0,C 180,E1 -465.921,E2 -465.921} C_VEL
LIN {X 0,Y 608.497,Z 263.491,A -85,B 0,C 180,E1 -468.723,E2 -468.723} C_VEL
LIN {X 0,Y 608.512,Z 247.074,A -85,B 0,C 180,E1 -471.157,E2 -471.157} C_VEL
LIN {X 0,Y 608.391,Z 239.51,A -85,B 0,C 180,E1 -472.319,E2 -472.319} C_VEL
LIN {X 0,Y 608.402,Z 239.507,A -85,B 0,C 180,E1 -474.574,E2 -474.574} C_VEL
LIN {X 0,Y 608.457,Z 239.507,A -85,B 0,C 180,E1 -477.203,E2 -477.203} C_VEL
LIN {X 0,Y 608.401,Z 239.508,A -85,B 0,C 180,E1 -479.961,E2 -479.961} C_VEL
LIN {X 0,Y 608.402,Z 239.507,A -85,B 0,C 180,E1 -482.514,E2 -482.514} C_VEL
LIN {X 0,Y 608.407,Z 239.516,A -85,B 0,C 180,E1 -485.28,E2 -485.28} C_VEL
LIN {X 0,Y 608.426,Z 239.505,A -85,B 0,C 180,E1 -487.75,E2 -487.75} C_VEL
LIN {X 0,Y 608.402,Z 239.507,A -85,B 0,C 180,E1 -490.323,E2 -490.323} C_VEL
LIN {X 0,Y 608.437,Z 239.511,A -85,B 0,C 180,E1 -492.961,E2 -492.961} C_VEL
LIN {X 0,Y 608.4,Z 239.507,A -85,B 0,C 180,E1 -495.742,E2 -495.742} C_VEL
LIN {X 0,Y 608.4,Z 239.507,A -85,B 0,C 180,E1 -497.934,E2 -497.934} C_VEL
LIN {X 0,Y 608.433,Z 239.509,A -85,B 0,C 180,E1 -500.707,E2 -500.707} C_VEL
LIN {X 0,Y 608.438,Z 239.509,A -85,B 0,C 180,E1 -503.084,E2 -503.084} C_VEL
LIN {X 0,Y 608.42,Z 239.505,A -85,B 0,C 180,E1 -505.528,E2 -505.528} C_VEL
LIN {X 0,Y 608.411,Z 239.505,A -85,B 0,C 180,E1 -507.902,E2 -507.902} C_VEL
LIN {X 0,Y 608.426,Z 239.506,A -85,B 0,C 180,E1 -510.218,E2 -510.218} C_VEL
LIN {X 0,Y 608.465,Z 239.507,A -85,B 0,C 180,E1 -512.795,E2 -512.795} C_VEL
LIN {X 0,Y 608.406,Z 239.506,A -85,B 0,C 180,E1 -515.427,E2 -515.427} C_VEL
LIN {X 0,Y 608.454,Z 239.506,A -85,B 0,C 180,E1 -518.308,E2 -518.308} C_VEL
LIN {X 0,Y 608.408,Z 239.506,A -85,B 0,C 180,E1 -521.302,E2 -521.302} C_VEL
LIN {X 0,Y 608.423,Z 239.506,A -85,B 0,C 180,E1 -523.905,E2 -523.905} C_VEL
LIN {X 0,Y 608.432,Z 239.509,A -85,B 0,C 180,E1 -526.643,E2 -526.643} C_VEL
LIN {X 0,Y 608.404,Z 239.506,A -85,B 0,C 180,E1 -529.349,E2 -529.349} C_VEL
LIN {X 0,Y 608.467,Z 239.505,A -85,B 0,C 180,E1 -532.033,E2 -532.033} C_VEL
LIN {X 0,Y 608.423,Z 239.507,A -85,B 0,C 180,E1 -534.698,E2 -534.698} C_VEL
LIN {X 0,Y 608.423,Z 239.504,A -85,B 0,C 180,E1 -537.352,E2 -537.352} C_VEL
LIN {X 0,Y 608.474,Z 239.506,A -85,B 0,C 180,E1 -540,E2 -540} C_VEL
LIN {X 0,Y 608.43,Z 239.505,A -85,B 0,C 180,E1 -542.648,E2 -542.648} C_VEL
LIN {X 0,Y 608.417,Z 239.505,A -85,B 0,C 180,E1 -545.302,E2 -545.302} C_VEL
LIN {X 0,Y 608.47,Z 239.509,A -85,B 0,C 180,E1 -547.967,E2 -547.967} C_VEL
LIN {X 0,Y 608.429,Z 239.505,A -85,B 0,C 180,E1 -549.416,E2 -549.416} C_VEL
LIN {X 0,Y 607.773,Z 239.595,A -85,B 0,C 180,E1 -549.968,E2 -549.968} C_VEL
LIN {X 0,Y 604.938,Z 239.948,A -85,B 0,C 180,E1 -550.865,E2 -550.865} C_VEL
LIN {X 0,Y 602.526,Z 240.248,A -85,B 0,C 180,E1 -551.587,E2 -551.587} C_VEL
LIN {X 0,Y 601.471,Z 240.376,A -85,B 0,C 180,E1 -552.143,E2 -552.143} C_VEL
LIN {X 0,Y 601.375,Z 240.385,A -85,B 0,C 180,E1 -552.331,E2 -552.331} C_VEL
LIN {X 0,Y 601.373,Z 240.382,A -85,B 0,C 180,E1 -554.898,E2 -554.898} C_VEL
LIN {X 0,Y 601.372,Z 240.392,A -85,B 0,C 180,E1 -557.689,E2 -557.689} C_VEL
LIN {X 0,Y 601.381,Z 240.39,A -85,B 0,C 180,E1 -559.81,E2 -559.81} C_VEL
LIN {X 0,Y 601.351,Z 240.385,A -85,B 0,C 180,E1 -562.59,E2 -562.59} C_VEL
LIN {X 0,Y 601.377,Z 240.382,A -85,B 0,C 180,E1 -564.88,E2 -564.88} C_VEL
LIN {X 0,Y 601.398,Z 240.386,A -85,B 0,C 180,E1 -567.359,E2 -567.359} C_VEL
LIN {X 0,Y 601.373,Z 240.383,A -85,B 0,C 180,E1 -570.167,E2 -570.167} C_VEL
LIN {X 0,Y 601.388,Z 240.381,A -85,B 0,C 180,E1 -572.71,E2 -572.71} C_VEL
LIN {X 0,Y 601.371,Z 240.388,A -85,B 0,C 180,E1 -575.108,E2 -575.108} C_VEL
LIN {X 0,Y 601.431,Z 240.384,A -85,B 0,C 180,E1 -577.419,E2 -577.419} C_VEL
LIN {X 0,Y 601.376,Z 240.383,A -85,B 0,C 180,E1 -579.998,E2 -579.998} C_VEL
LIN {X 0,Y 601.372,Z 240.384,A -85,B 0,C 180,E1 -582.674,E2 -582.674} C_VEL
LIN {X 0,Y 601.4,Z 240.384,A -85,B 0,C 180,E1 -585.479,E2 -585.479} C_VEL
LIN {X 0,Y 601.404,Z 240.379,A -85,B 0,C 180,E1 -588.409,E2 -588.409} C_VEL
LIN {X 0,Y 601.4,Z 240.386,A -85,B 0,C 180,E1 -590.872,E2 -590.872} C_VEL
LIN {X 0,Y 601.396,Z 240.383,A -85,B 0,C 180,E1 -593.416,E2 -593.416} C_VEL
LIN {X 0,Y 601.4,Z 240.379,A -85,B 0,C 180,E1 -596.069,E2 -596.069} C_VEL
LIN {X 0,Y 601.395,Z 240.387,A -85,B 0,C 180,E1 -599.056,E2 -599.056} C_VEL
LIN {X 0,Y 601.394,Z 240.382,A -85,B 0,C 180,E1 -601.371,E2 -601.371} C_VEL
LIN {X 0,Y 601.377,Z 240.382,A -85,B 0,C 180,E1 -603.635,E2 -603.635} C_VEL
LIN {X 0,Y 601.396,Z 240.379,A -85,B 0,C 180,E1 -605.857,E2 -605.857} C_VEL
LIN {X 0,Y 601.395,Z 240.389,A -85,B 0,C 180,E1 -608.76,E2 -608.76} C_VEL
LIN {X 0,Y 601.363,Z 240.383,A -85,B 0,C 180,E1 -611.606,E2 -611.606} C_VEL
LIN {X 0,Y 601.433,Z 240.443,A -85,B 0,C 180,E1 -614.148,E2 -614.148} C_VEL
LIN {X 0,Y 601.36,Z 252.301,A -85,B 0,C 180,E1 -616.827,E2 -616.827} C_VEL
LIN {X 0,Y 601.294,Z 263.012,A -85,B 0,C 180,E1 -619.221,E2 -619.221} C_VEL
LIN {X 0,Y 601.335,Z 265.211,A -85,B 0,C 180,E1 -619.712,E2 -619.712} C_VEL
LIN {X 0,Y 601.512,Z 300.834,A -85,B 0,C 180,E1 -620.14,E2 -620.14} C_VEL
LIN {X 0,Y 601.453,Z 340.264,A -85,B 0,C 180,E1 -620.627,E2 -620.627} C_VEL
LIN {X 0,Y 601.454,Z 349.961,A -85,B 0,C 180,E1 -620.839,E2 -620.839} C_VEL
LIN {X 0,Y 601.4,Z 361.543,A -85,B 0,C 180,E1 -621.219,E2 -621.219} C_VEL
LIN {X 0,Y 601.443,Z 371.436,A -85,B 0,C 180,E1 -621.685,E2 -621.685} C_VEL
LIN {X 0,Y 601.412,Z 379.892,A -85,B 0,C 180,E1 -622.192,E2 -622.192} C_VEL
LIN {X 0,Y 601.411,Z 387.858,A -85,B 0,C 180,E1 -622.783,E2 -622.783} C_VEL
LIN {X 0,Y 601.413,Z 395.146,A -85,B 0,C 180,E1 -623.443,E2 -623.443} C_VEL
LIN {X 0,Y 601.386,Z 401.398,A -85,B 0,C 180,E1 -624.131,E2 -624.131} C_VEL
LIN {X 0,Y 601.347,Z 407.642,A -85,B 0,C 180,E1 -624.971,E2 -624.971} C_VEL
LIN {X 0,Y 601.345,Z 413.426,A -85,B 0,C 180,E1 -625.979,E2 -625.979} C_VEL
LIN {X 0,Y 601.345,Z 417.632,A -85,B 0,C 180,E1 -626.985,E2 -626.985} C_VEL
LIN {X 0,Y 601.343,Z 420.571,A -85,B 0,C 180,E1 -627.99,E2 -627.99} C_VEL
LIN {X 0,Y 601.345,Z 421.871,A -85,B 0,C 180,E1 -628.66,E2 -628.66} C_VEL
LIN {X 0,Y 601.335,Z 422.692,A -85,B 0,C 180,E1 -629.33,E2 -629.33} C_VEL
LIN {X 0,Y 601.333,Z 422.995,A -85,B 0,C 180,E1 -630,E2 -630} C_VEL
LIN {X 0,Y 601.336,Z 422.735,A -85,B 0,C 180,E1 -630.669,E2 -630.669} C_VEL
LIN {X 0,Y 601.346,Z 421.998,A -85,B 0,C 180,E1 -631.339,E2 -631.339} C_VEL
LIN {X 0,Y 601.343,Z 420.787,A -85,B 0,C 180,E1 -632.009,E2 -632.009} C_VEL
LIN {X 0,Y 601.344,Z 417.942,A -85,B 0,C 180,E1 -633.014,E2 -633.014} C_VEL
LIN {X 0,Y 601.365,Z 415.351,A -85,B 0,C 180,E1 -633.685,E2 -633.685} C_VEL
LIN {X 0,Y 601.362,Z 410.244,A -85,B 0,C 180,E1 -634.692,E2 -634.692} C_VEL
LIN {X 0,Y 601.384,Z 404.748,A -85,B 0,C 180,E1 -635.532,E2 -635.532} C_VEL
LIN {X 0,Y 601.394,Z 396.589,A -85,B 0,C 180,E1 -636.504,E2 -636.504} C_VEL
LIN {X 0,Y 601.413,Z 388.947,A -85,B 0,C 180,E1 -637.216,E2 -637.216} C_VEL
LIN {X 0,Y 601.412,Z 381.198,A -85,B 0,C 180,E1 -637.807,E2 -637.807} C_VEL
LIN {X 0,Y 601.45,Z 373.034,A -85,B 0,C 180,E1 -638.314,E2 -638.314} C_VEL
LIN {X 0,Y 601.399,Z 362.667,A -85,B 0,C 180,E1 -638.822,E2 -638.822} C_VEL
LIN {X 0,Y 601.436,Z 351.022,A -85,B 0,C 180,E1 -639.224,E2 -639.224} C_VEL
LIN {X 0,Y 601.462,Z 340.627,A -85,B 0,C 180,E1 -639.457,E2 -639.457} C_VEL
LIN {X 0,Y 601.531,Z 292.374,A -85,B 0,C 180,E1 -640.05,E2 -640.05} C_VEL
LIN {X 0,Y 601.363,Z 265.539,A -85,B 0,C 180,E1 -640.372,E2 -640.372} C_VEL
LIN {X 0,Y 601.317,Z 264.949,A -85,B 0,C 180,E1 -640.437,E2 -640.437} C_VEL
LIN {X 0,Y 601.35,Z 252.705,A -85,B 0,C 180,E1 -643.173,E2 -643.173} C_VEL
LIN {X 0,Y 601.404,Z 240.381,A -85,B 0,C 180,E1 -645.982,E2 -645.982} C_VEL
LIN {X 0,Y 601.401,Z 240.384,A -85,B 0,C 180,E1 -649.099,E2 -649.099} C_VEL
LIN {X 0,Y 601.377,Z 240.383,A -85,B 0,C 180,E1 -651.96,E2 -651.96} C_VEL
LIN {X 0,Y 601.377,Z 240.385,A -85,B 0,C 180,E1 -654.879,E2 -654.879} C_VEL
LIN {X 0,Y 601.403,Z 240.387,A -85,B 0,C 180,E1 -657.36,E2 -657.36} C_VEL
LIN {X 0,Y 601.369,Z 240.383,A -85,B 0,C 180,E1 -660.167,E2 -660.167} C_VEL
LIN {X 0,Y 601.388,Z 240.384,A -85,B 0,C 180,E1 -662.71,E2 -662.71} C_VEL
LIN {X 0,Y 601.37,Z 240.393,A -85,B 0,C 180,E1 -665.108,E2 -665.108} C_VEL
LIN {X 0,Y 601.427,Z 240.38,A -85,B 0,C 180,E1 -667.419,E2 -667.419} C_VEL
LIN {X 0,Y 601.371,Z 240.382,A -85,B 0,C 180,E1 -669.998,E2 -669.998} C_VEL
LIN {X 0,Y 601.372,Z 240.388,A -85,B 0,C 180,E1 -672.673,E2 -672.673} C_VEL
LIN {X 0,Y 601.395,Z 240.381,A -85,B 0,C 180,E1 -675.479,E2 -675.479} C_VEL
LIN {X 0,Y 601.402,Z 240.382,A -85,B 0,C 180,E1 -678.408,E2 -678.408} C_VEL
LIN {X 0,Y 601.393,Z 240.388,A -85,B 0,C 180,E1 -680.872,E2 -680.872} C_VEL
LIN {X 0,Y 601.383,Z 240.382,A -85,B 0,C 180,E1 -683.415,E2 -683.415} C_VEL
LIN {X 0,Y 601.392,Z 240.382,A -85,B 0,C 180,E1 -686.069,E2 -686.069} C_VEL
LIN {X 0,Y 601.384,Z 240.384,A -85,B 0,C 180,E1 -689.056,E2 -689.056} C_VEL
LIN {X 0,Y 601.38,Z 240.381,A -85,B 0,C 180,E1 -691.37,E2 -691.37} C_VEL
LIN {X 0,Y 601.393,Z 240.384,A -85,B 0,C 180,E1 -694.135,E2 -694.135} C_VEL
LIN {X 0,Y 601.37,Z 240.39,A -85,B 0,C 180,E1 -696.588,E2 -696.588} C_VEL
LIN {X 0,Y 601.383,Z 240.381,A -85,B 0,C 180,E1 -699.476,E2 -699.476} C_VEL
LIN {X 0,Y 601.358,Z 240.385,A -85,B 0,C 180,E1 -701.606,E2 -701.606} C_VEL
LIN {X 0,Y 601.382,Z 240.389,A -85,B 0,C 180,E1 -704.408,E2 -704.408} C_VEL
LIN {X 0,Y 601.387,Z 240.386,A -85,B 0,C 180,E1 -706.483,E2 -706.483} C_VEL
LIN {X 0,Y 601.349,Z 240.385,A -85,B 0,C 180,E1 -709.223,E2 -709.223} C_VEL
LIN {X 0,Y 601.424,Z 240.384,A -85,B 0,C 180,E1 -711.939,E2 -711.939} C_VEL
LIN {X 0,Y 601.386,Z 240.382,A -85,B 0,C 180,E1 -714.635,E2 -714.635} C_VEL
LIN {X 0,Y 601.392,Z 240.381,A -85,B 0,C 180,E1 -717.321,E2 -717.321} C_VEL
LIN {X 0,Y 601.438,Z 240.383,A -85,B 0,C 180,E1 -720,E2 -720} C_VEL
LIN {X 0,Y 601.389,Z 240.381,A -85,B 0,C 180,E1 -722.679,E2 -722.679} C_VEL
LIN {X 0,Y 601.388,Z 240.383,A -85,B 0,C 180,E1 -725.364,E2 -725.364} C_VEL
LIN {X 0,Y 601.422,Z 240.381,A -85,B 0,C 180,E1 -728.061,E2 -728.061} C_VEL
LIN {X 0,Y 601.37,Z 240.383,A -85,B 0,C 180,E1 -730.988,E2 -730.988} C_VEL
LIN {X 0,Y 601.382,Z 240.389,A -85,B 0,C 180,E1 -733.517,E2 -733.517} C_VEL
LIN {X 0,Y 601.381,Z 240.382,A -85,B 0,C 180,E1 -736.288,E2 -736.288} C_VEL
LIN {X 0,Y 601.394,Z 240.383,A -85,B 0,C 180,E1 -739.1,E2 -739.1} C_VEL
LIN {X 0,Y 601.371,Z 240.385,A -85,B 0,C 180,E1 -741.961,E2 -741.961} C_VEL
LIN {X 0,Y 601.368,Z 240.385,A -85,B 0,C 180,E1 -744.88,E2 -744.88} C_VEL
LIN {X 0,Y 601.393,Z 240.39,A -85,B 0,C 180,E1 -747.36,E2 -747.36} C_VEL
LIN {X 0,Y 601.364,Z 240.383,A -85,B 0,C 180,E1 -750.167,E2 -750.167} C_VEL
LIN {X 0,Y 601.38,Z 240.384,A -85,B 0,C 180,E1 -752.71,E2 -752.71} C_VEL
LIN {X 0,Y 601.363,Z 240.393,A -85,B 0,C 180,E1 -755.108,E2 -755.108} C_VEL
LIN {X 0,Y 601.422,Z 240.381,A -85,B 0,C 180,E1 -757.42,E2 -757.42} C_VEL
LIN {X 0,Y 601.368,Z 240.383,A -85,B 0,C 180,E1 -759.998,E2 -759.998} C_VEL
LIN {X 0,Y 601.363,Z 240.388,A -85,B 0,C 180,E1 -762.675,E2 -762.675} C_VEL
LIN {X 0,Y 601.394,Z 240.382,A -85,B 0,C 180,E1 -765.48,E2 -765.48} C_VEL
LIN {X 0,Y 601.395,Z 240.382,A -85,B 0,C 180,E1 -768.41,E2 -768.41} C_VEL
LIN {X 0,Y 601.39,Z 240.39,A -85,B 0,C 180,E1 -770.872,E2 -770.872} C_VEL
LIN {X 0,Y 601.369,Z 240.384,A -85,B 0,C 180,E1 -773.415,E2 -773.415} C_VEL
LIN {X 0,Y 601.377,Z 240.383,A -85,B 0,C 180,E1 -776.072,E2 -776.072} C_VEL
LIN {X 0,Y 601.381,Z 240.385,A -85,B 0,C 180,E1 -779.056,E2 -779.056} C_VEL
LIN {X 0,Y 601.375,Z 240.383,A -85,B 0,C 180,E1 -781.371,E2 -781.371} C_VEL
LIN {X 0,Y 601.382,Z 240.385,A -85,B 0,C 180,E1 -784.139,E2 -784.139} C_VEL
LIN {X 0,Y 601.363,Z 240.394,A -85,B 0,C 180,E1 -786.588,E2 -786.588} C_VEL
LIN {X 0,Y 601.374,Z 240.567,A -85,B 0,C 180,E1 -787.59,E2 -787.59} C_VEL
LIN {X 0,Y 601.584,Z 248.266,A -85,B 0,C 180,E1 -788.768,E2 -788.768} C_VEL
LIN {X 0,Y 601.509,Z 265.721,A -85,B 0,C 180,E1 -791.383,E2 -791.383} C_VEL
LIN {X 0,Y 601.49,Z 285.059,A -85,B 0,C 180,E1 -794.237,E2 -794.237} C_VEL
LIN {X 0,Y 601.436,Z 304.048,A -85,B 0,C 180,E1 -797.001,E2 -797.001} C_VEL
LIN {X 0,Y 601.366,Z 322.296,A -85,B 0,C 180,E1 -799.628,E2 -799.628} C_VEL
LIN {X 0,Y 601.468,Z 400.466,A -85,B 0,C 180,E1 -800.585,E2 -800.585} C_VEL
LIN {X 0,Y 601.431,Z 410.92,A -85,B 0,C 180,E1 -800.818,E2 -800.818} C_VEL
LIN {X 0,Y 601.412,Z 423.545,A -85,B 0,C 180,E1 -801.262,E2 -801.262} C_VEL
LIN {X 0,Y 601.45,Z 432.242,A -85,B 0,C 180,E1 -801.686,E2 -801.686} C_VEL
LIN {X 0,Y 601.412,Z 440.549,A -85,B 0,C 180,E1 -802.193,E2 -802.193} C_VEL
LIN {X 0,Y 601.411,Z 448.406,A -85,B 0,C 180,E1 -802.784,E2 -802.784} C_VEL
LIN {X 0,Y 601.411,Z 455.599,A -85,B 0,C 180,E1 -803.443,E2 -803.443} C_VEL
LIN {X 0,Y 601.391,Z 463.194,A -85,B 0,C 180,E1 -804.3,E2 -804.3} C_VEL
LIN {X 0,Y 601.38,Z 469.03,A -85,B 0,C 180,E1 -805.14,E2 -805.14} C_VEL
LIN {X 0,Y 601.345,Z 473.633,A -85,B 0,C 180,E1 -805.979,E2 -805.979} C_VEL
LIN {X 0,Y 601.343,Z 476.623,A -85,B 0,C 180,E1 -806.65,E2 -806.65} C_VEL
LIN {X 0,Y 601.326,Z 478.933,A -85,B 0,C 180,E1 -807.321,E2 -807.321} C_VEL
LIN {X 0,Y 601.343,Z 480.68,A -85,B 0,C 180,E1 -807.991,E2 -807.991} C_VEL
LIN {X 0,Y 601.345,Z 481.935,A -85,B 0,C 180,E1 -808.661,E2 -808.661} C_VEL
LIN {X 0,Y 601.335,Z 482.714,A -85,B 0,C 180,E1 -809.331,E2 -809.331} C_VEL
LIN {X 0,Y 601.332,Z 483,A -85,B 0,C 180,E1 -810,E2 -810} C_VEL
LIN {X 0,Y 601.335,Z 482.713,A -85,B 0,C 180,E1 -810.67,E2 -810.67} C_VEL
LIN {X 0,Y 601.345,Z 481.934,A -85,B 0,C 180,E1 -811.34,E2 -811.34} C_VEL
LIN {X 0,Y 601.343,Z 480.678,A -85,B 0,C 180,E1 -812.01,E2 -812.01} C_VEL
LIN {X 0,Y 601.342,Z 477.785,A -85,B 0,C 180,E1 -813.015,E2 -813.015} C_VEL
LIN {X 0,Y 601.364,Z 475.145,A -85,B 0,C 180,E1 -813.686,E2 -813.686} C_VEL
LIN {X 0,Y 601.341,Z 469.983,A -85,B 0,C 180,E1 -814.693,E2 -814.693} C_VEL
LIN {X 0,Y 601.383,Z 464.428,A -85,B 0,C 180,E1 -815.533,E2 -815.533} C_VEL
LIN {X 0,Y 601.393,Z 457.151,A -85,B 0,C 180,E1 -816.403,E2 -816.403} C_VEL
LIN {X 0,Y 601.414,Z 449.412,A -85,B 0,C 180,E1 -817.133,E2 -817.133} C_VEL
LIN {X 0,Y 601.433,Z 441.758,A -85,B 0,C 180,E1 -817.723,E2 -817.723} C_VEL
LIN {X 0,Y 601.443,Z 433.717,A -85,B 0,C 180,E1 -818.23,E2 -818.23} C_VEL
LIN {X 0,Y 601.426,Z 425.385,A -85,B 0,C 180,E1 -818.653,E2 -818.653} C_VEL
LIN {X 0,Y 601.421,Z 416.881,A -85,B 0,C 180,E1 -818.992,E2 -818.992} C_VEL
LIN {X 0,Y 601.45,Z 406.742,A -85,B 0,C 180,E1 -819.288,E2 -819.288} C_VEL
LIN {X 0,Y 601.484,Z 395.032,A -85,B 0,C 180,E1 -819.5,E2 -819.5} C_VEL
LIN {X 0,Y 601.366,Z 322.291,A -85,B 0,C 180,E1 -820.373,E2 -820.373} C_VEL
LIN {X 0,Y 601.437,Z 304.043,A -85,B 0,C 180,E1 -823,E2 -823} C_VEL
LIN {X 0,Y 601.484,Z 283.867,A -85,B 0,C 180,E1 -825.938,E2 -825.938} C_VEL
LIN {X 0,Y 601.509,Z 265.717,A -85,B 0,C 180,E1 -828.617,E2 -828.617} C_VEL
LIN {X 0,Y 601.585,Z 248.261,A -85,B 0,C 180,E1 -831.233,E2 -831.233} C_VEL
LIN {X 0,Y 601.362,Z 240.396,A -85,B 0,C 180,E1 -832.436,E2 -832.436} C_VEL
LIN {X 0,Y 601.367,Z 240.385,A -85,B 0,C 180,E1 -834.88,E2 -834.88} C_VEL
LIN {X 0,Y 601.392,Z 240.39,A -85,B 0,C 180,E1 -837.358,E2 -837.358} C_VEL
LIN {X 0,Y 601.368,Z 240.383,A -85,B 0,C 180,E1 -840.168,E2 -840.168} C_VEL
LIN {X 0,Y 601.379,Z 240.383,A -85,B 0,C 180,E1 -842.709,E2 -842.709} C_VEL
LIN {X 0,Y 601.362,Z 240.392,A -85,B 0,C 180,E1 -845.107,E2 -845.107} C_VEL
LIN {X 0,Y 601.398,Z 240.385,A -85,B 0,C 180,E1 -847.422,E2 -847.422} C_VEL
LIN {X 0,Y 601.364,Z 240.383,A -85,B 0,C 180,E1 -849.999,E2 -849.999} C_VEL
LIN {X 0,Y 601.362,Z 240.387,A -85,B 0,C 180,E1 -852.675,E2 -852.675} C_VEL
LIN {X 0,Y 601.399,Z 240.382,A -85,B 0,C 180,E1 -855.48,E2 -855.48} C_VEL
LIN {X 0,Y 601.382,Z 240.383,A -85,B 0,C 180,E1 -858.412,E2 -858.412} C_VEL
LIN {X 0,Y 601.393,Z 240.389,A -85,B 0,C 180,E1 -860.872,E2 -860.872} C_VEL
LIN {X 0,Y 601.375,Z 240.384,A -85,B 0,C 180,E1 -863.415,E2 -863.415} C_VEL
LIN {X 0,Y 601.381,Z 240.382,A -85,B 0,C 180,E1 -866.072,E2 -866.072} C_VEL
LIN {X 0,Y 601.388,Z 240.387,A -85,B 0,C 180,E1 -868.551,E2 -868.551} C_VEL
LIN {X 0,Y 601.38,Z 240.382,A -85,B 0,C 180,E1 -871.371,E2 -871.371} C_VEL
LIN {X 0,Y 601.366,Z 240.383,A -85,B 0,C 180,E1 -873.635,E2 -873.635} C_VEL
LIN {X 0,Y 601.387,Z 240.381,A -85,B 0,C 180,E1 -875.857,E2 -875.857} C_VEL
LIN {X 0,Y 601.389,Z 240.387,A -85,B 0,C 180,E1 -878.76,E2 -878.76} C_VEL
LIN {X 0,Y 601.355,Z 240.384,A -85,B 0,C 180,E1 -881.606,E2 -881.606} C_VEL
LIN {X 0,Y 601.385,Z 240.391,A -85,B 0,C 180,E1 -884.408,E2 -884.408} C_VEL
LIN {X 0,Y 601.352,Z 240.385,A -85,B 0,C 180,E1 -887.17,E2 -887.17} C_VEL
LIN {X 0,Y 601.415,Z 240.38,A -85,B 0,C 180,E1 -889.905,E2 -889.905} C_VEL
LIN {X 0,Y 601.374,Z 240.387,A -85,B 0,C 180,E1 -892.614,E2 -892.614} C_VEL
LIN {X 0,Y 601.37,Z 240.383,A -85,B 0,C 180,E1 -895.308,E2 -895.308} C_VEL
LIN {X 0,Y 601.433,Z 240.382,A -85,B 0,C 180,E1 -897.991,E2 -897.991} C_VEL
LIN {X 0,Y 601.367,Z 240.385,A -85,B 0,C 180,E1 -900.67,E2 -900.67} C_VEL
LIN {X 0,Y 601.398,Z 240.381,A -85,B 0,C 180,E1 -902.679,E2 -902.679} C_VEL
LIN {X 0,Y 601.387,Z 240.382,A -85,B 0,C 180,E1 -905.365,E2 -905.365} C_VEL
LIN {X 0,Y 601.429,Z 240.384,A -85,B 0,C 180,E1 -908.061,E2 -908.061} C_VEL
LIN {X 0,Y 601.376,Z 240.382,A -85,B 0,C 180,E1 -910.987,E2 -910.987} C_VEL
LIN {X 0,Y 601.375,Z 240.385,A -85,B 0,C 180,E1 -912.331,E2 -912.331} C_VEL
LIN {X 0,Y 600.684,Z 240.471,A -85,B 0,C 180,E1 -912.891,E2 -912.891} C_VEL
LIN {X 0,Y 597.829,Z 240.834,A -85,B 0,C 180,E1 -913.799,E2 -913.799} C_VEL
LIN {X 0,Y 595.433,Z 241.127,A -85,B 0,C 180,E1 -914.529,E2 -914.529} C_VEL
LIN {X 0,Y 594.407,Z 241.251,A -85,B 0,C 180,E1 -915.093,E2 -915.093} C_VEL
LIN {X 0,Y 594.323,Z 241.263,A -85,B 0,C 180,E1 -915.283,E2 -915.283} C_VEL
LIN {X 0,Y 594.322,Z 241.268,A -85,B 0,C 180,E1 -917.906,E2 -917.906} C_VEL
LIN {X 0,Y 594.37,Z 241.255,A -85,B 0,C 180,E1 -920.777,E2 -920.777} C_VEL
LIN {X 0,Y 594.344,Z 241.267,A -85,B 0,C 180,E1 -923.706,E2 -923.706} C_VEL
LIN {X 0,Y 594.351,Z 241.261,A -85,B 0,C 180,E1 -926.015,E2 -926.015} C_VEL
LIN {X 0,Y 594.341,Z 241.26,A -85,B 0,C 180,E1 -928.95,E2 -928.95} C_VEL
LIN {X 0,Y 594.366,Z 241.263,A -85,B 0,C 180,E1 -931.641,E2 -931.641} C_VEL
LIN {X 0,Y 594.357,Z 241.257,A -85,B 0,C 180,E1 -934.135,E2 -934.135} C_VEL
LIN {X 0,Y 594.377,Z 241.26,A -85,B 0,C 180,E1 -937.087,E2 -937.087} C_VEL
LIN {X 0,Y 594.337,Z 241.262,A -85,B 0,C 180,E1 -939.77,E2 -939.77} C_VEL
LIN {X 0,Y 594.332,Z 241.26,A -85,B 0,C 180,E1 -942.379,E2 -942.379} C_VEL
LIN {X 0,Y 594.339,Z 241.268,A -85,B 0,C 180,E1 -945.194,E2 -945.194} C_VEL
LIN {X 0,Y 594.357,Z 241.256,A -85,B 0,C 180,E1 -948.155,E2 -948.155} C_VEL
LIN {X 0,Y 594.364,Z 241.262,A -85,B 0,C 180,E1 -951.298,E2 -951.298} C_VEL
LIN {X 0,Y 594.339,Z 241.259,A -85,B 0,C 180,E1 -953.754,E2 -953.754} C_VEL
LIN {X 0,Y 594.351,Z 241.258,A -85,B 0,C 180,E1 -956.237,E2 -956.237} C_VEL
LIN {X 0,Y 594.346,Z 241.263,A -85,B 0,C 180,E1 -958.648,E2 -958.648} C_VEL
LIN {X 0,Y 594.371,Z 241.262,A -85,B 0,C 180,E1 -961.045,E2 -961.045} C_VEL
LIN {X 0,Y 594.363,Z 241.258,A -85,B 0,C 180,E1 -963.299,E2 -963.299} C_VEL
LIN {X 0,Y 594.334,Z 241.26,A -85,B 0,C 180,E1 -965.578,E2 -965.578} C_VEL
LIN {X 0,Y 594.351,Z 241.264,A -85,B 0,C 180,E1 -968.496,E2 -968.496} C_VEL
LIN {X 0,Y 594.345,Z 241.259,A -85,B 0,C 180,E1 -971.381,E2 -971.381} C_VEL
LIN {X 0,Y 594.387,Z 241.402,A -85,B 0,C 180,E1 -974.175,E2 -974.175} C_VEL
LIN {X 0,Y 594.269,Z 253.834,A -85,B 0,C 180,E1 -977.014,E2 -977.014} C_VEL
LIN {X 0,Y 594.253,Z 265.214,A -85,B 0,C 180,E1 -979.588,E2 -979.588} C_VEL
LIN {X 0,Y 594.558,Z 274.052,A -85,B 0,C 180,E1 -979.701,E2 -979.701} C_VEL
LIN {X 0,Y 594.468,Z 340.296,A -85,B 0,C 180,E1 -980.516,E2 -980.516} C_VEL
LIN {X 0,Y 594.451,Z 349.982,A -85,B 0,C 180,E1 -980.73,E2 -980.73} C_VEL
LIN {X 0,Y 594.386,Z 361.556,A -85,B 0,C 180,E1 -981.115,E2 -981.115} C_VEL
LIN {X 0,Y 594.408,Z 371.442,A -85,B 0,C 180,E1 -981.586,E2 -981.586} C_VEL
LIN {X 0,Y 594.37,Z 379.9,A -85,B 0,C 180,E1 -982.099,E2 -982.099} C_VEL
LIN {X 0,Y 594.353,Z 387.866,A -85,B 0,C 180,E1 -982.697,E2 -982.697} C_VEL
LIN {X 0,Y 594.344,Z 395.067,A -85,B 0,C 180,E1 -983.357,E2 -983.357} C_VEL
LIN {X 0,Y 594.318,Z 402.82,A -85,B 0,C 180,E1 -984.231,E2 -984.231} C_VEL
LIN {X 0,Y 594.255,Z 409.73,A -85,B 0,C 180,E1 -985.251,E2 -985.251} C_VEL
LIN {X 0,Y 594.287,Z 414.945,A -85,B 0,C 180,E1 -986.27,E2 -986.27} C_VEL
LIN {X 0,Y 594.248,Z 417.634,A -85,B 0,C 180,E1 -986.949,E2 -986.949} C_VEL
LIN {X 0,Y 594.242,Z 420.573,A -85,B 0,C 180,E1 -987.966,E2 -987.966} C_VEL
LIN {X 0,Y 594.244,Z 421.872,A -85,B 0,C 180,E1 -988.644,E2 -988.644} C_VEL
LIN {X 0,Y 594.235,Z 422.691,A -85,B 0,C 180,E1 -989.322,E2 -989.322} C_VEL
LIN {X 0,Y 594.234,Z 422.996,A -85,B 0,C 180,E1 -990,E2 -990} C_VEL
LIN {X 0,Y 594.236,Z 422.734,A -85,B 0,C 180,E1 -990.677,E2 -990.677} C_VEL
LIN {X 0,Y 594.246,Z 421.998,A -85,B 0,C 180,E1 -991.355,E2 -991.355} C_VEL
LIN {X 0,Y 594.242,Z 420.787,A -85,B 0,C 180,E1 -992.033,E2 -992.033} C_VEL
LIN {X 0,Y 594.247,Z 417.941,A -85,B 0,C 180,E1 -993.05,E2 -993.05} C_VEL
LIN {X 0,Y 594.286,Z 415.35,A -85,B 0,C 180,E1 -993.729,E2 -993.729} C_VEL
LIN {X 0,Y 594.265,Z 410.242,A -85,B 0,C 180,E1 -994.748,E2 -994.748} C_VEL
LIN {X 0,Y 594.31,Z 404.745,A -85,B 0,C 180,E1 -995.598,E2 -995.598} C_VEL
LIN {X 0,Y 594.342,Z 397.617,A -85,B 0,C 180,E1 -996.476,E2 -996.476} C_VEL
LIN {X 0,Y 594.354,Z 388.941,A -85,B 0,C 180,E1 -997.302,E2 -997.302} C_VEL
LIN {X 0,Y 594.378,Z 381.193,A -85,B 0,C 180,E1 -997.9,E2 -997.9} C_VEL
LIN {X 0,Y 594.422,Z 373.028,A -85,B 0,C 180,E1 -998.413,E2 -998.413} C_VEL
LIN {X 0,Y 594.391,Z 362.652,A -85,B 0,C 180,E1 -998.927,E2 -998.927} C_VEL
LIN {X 0,Y 594.431,Z 351.001,A -85,B 0,C 180,E1 -999.334,E2 -999.334} C_VEL
LIN {X 0,Y 594.477,Z 340.594,A -85,B 0,C 180,E1 -999.569,E2 -999.569} C_VEL
LIN {X 0,Y 594.557,Z 290.54,A -85,B 0,C 180,E1 -1000.191,E2 -1000.191} C_VEL
LIN {X 0,Y 594.428,Z 266.501,A -85,B 0,C 180,E1 -1000.482,E2 -1000.482} C_VEL
LIN {X 0,Y 594.238,Z 265.138,A -85,B 0,C 180,E1 -1000.52,E2 -1000.52} C_VEL
LIN {X 0,Y 594.299,Z 252.702,A -85,B 0,C 180,E1 -1003.332,E2 -1003.332} C_VEL
LIN {X 0,Y 594.344,Z 241.262,A -85,B 0,C 180,E1 -1005.957,E2 -1005.957} C_VEL
LIN {X 0,Y 594.353,Z 241.259,A -85,B 0,C 180,E1 -1008.92,E2 -1008.92} C_VEL
LIN {X 0,Y 594.345,Z 241.266,A -85,B 0,C 180,E1 -1011.504,E2 -1011.504} C_VEL
LIN {X 0,Y 594.339,Z 241.259,A -85,B 0,C 180,E1 -1014.448,E2 -1014.448} C_VEL
LIN {X 0,Y 594.356,Z 241.258,A -85,B 0,C 180,E1 -1016.7,E2 -1016.7} C_VEL
LIN {X 0,Y 594.332,Z 241.261,A -85,B 0,C 180,E1 -1019.778,E2 -1019.778} C_VEL
LIN {X 0,Y 594.335,Z 241.259,A -85,B 0,C 180,E1 -1022.149,E2 -1022.149} C_VEL
LIN {X 0,Y 594.354,Z 241.259,A -85,B 0,C 180,E1 -1024.581,E2 -1024.581} C_VEL
LIN {X 0,Y 594.377,Z 241.256,A -85,B 0,C 180,E1 -1027.607,E2 -1027.607} C_VEL
LIN {X 0,Y 594.336,Z 241.263,A -85,B 0,C 180,E1 -1030.569,E2 -1030.569} C_VEL
LIN {X 0,Y 594.338,Z 241.263,A -85,B 0,C 180,E1 -1033.301,E2 -1033.301} C_VEL
LIN {X 0,Y 594.338,Z 241.26,A -85,B 0,C 180,E1 -1036.163,E2 -1036.163} C_VEL
LIN {X 0,Y 594.355,Z 241.261,A -85,B 0,C 180,E1 -1039.18,E2 -1039.18} C_VEL
LIN {X 0,Y 594.343,Z 241.259,A -85,B 0,C 180,E1 -1042.056,E2 -1042.056} C_VEL
LIN {X 0,Y 594.313,Z 241.272,A -85,B 0,C 180,E1 -1044.681,E2 -1044.681} C_VEL
LIN {X 0,Y 594.364,Z 241.259,A -85,B 0,C 180,E1 -1047.09,E2 -1047.09} C_VEL
LIN {X 0,Y 594.341,Z 241.258,A -85,B 0,C 180,E1 -1049.678,E2 -1049.678} C_VEL
LIN {X 0,Y 594.353,Z 241.267,A -85,B 0,C 180,E1 -1052.538,E2 -1052.538} C_VEL
LIN {X 0,Y 594.357,Z 241.261,A -85,B 0,C 180,E1 -1054.806,E2 -1054.806} C_VEL
LIN {X 0,Y 594.301,Z 241.263,A -85,B 0,C 180,E1 -1057.278,E2 -1057.278} C_VEL
LIN {X 0,Y 594.341,Z 241.262,A -85,B 0,C 180,E1 -1059.945,E2 -1059.945} C_VEL
LIN {X 0,Y 594.316,Z 241.264,A -85,B 0,C 180,E1 -1062.804,E2 -1062.804} C_VEL
LIN {X 0,Y 594.344,Z 241.26,A -85,B 0,C 180,E1 -1065.622,E2 -1065.622} C_VEL
LIN {X 0,Y 594.363,Z 241.262,A -85,B 0,C 180,E1 -1068.404,E2 -1068.404} C_VEL
LIN {X 0,Y 594.32,Z 241.261,A -85,B 0,C 180,E1 -1071.157,E2 -1071.157} C_VEL
LIN {X 0,Y 594.374,Z 241.262,A -85,B 0,C 180,E1 -1073.891,E2 -1073.891} C_VEL
LIN {X 0,Y 594.309,Z 241.264,A -85,B 0,C 180,E1 -1076.61,E2 -1076.61} C_VEL
LIN {X 0,Y 594.331,Z 241.261,A -85,B 0,C 180,E1 -1078.645,E2 -1078.645} C_VEL
LIN {X 0,Y 594.314,Z 241.262,A -85,B 0,C 180,E1 -1080.677,E2 -1080.677} C_VEL
LIN {X 0,Y 594.357,Z 241.256,A -85,B 0,C 180,E1 -1082.711,E2 -1082.711} C_VEL
LIN {X 0,Y 594.358,Z 241.26,A -85,B 0,C 180,E1 -1085.428,E2 -1085.428} C_VEL
LIN {X 0,Y 594.364,Z 241.259,A -85,B 0,C 180,E1 -1088.157,E2 -1088.157} C_VEL
LIN {X 0,Y 594.339,Z 241.26,A -85,B 0,C 180,E1 -1091.051,E2 -1091.051} C_VEL
LIN {X 0,Y 594.349,Z 241.267,A -85,B 0,C 180,E1 -1093.68,E2 -1093.68} C_VEL
LIN {X 0,Y 594.312,Z 241.262,A -85,B 0,C 180,E1 -1096.695,E2 -1096.695} C_VEL
LIN {X 0,Y 594.345,Z 241.265,A -85,B 0,C 180,E1 -1099.335,E2 -1099.335} C_VEL
LIN {X 0,Y 594.339,Z 241.269,A -85,B 0,C 180,E1 -1101.504,E2 -1101.504} C_VEL
LIN {X 0,Y 594.333,Z 241.259,A -85,B 0,C 180,E1 -1104.448,E2 -1104.448} C_VEL
LIN {X 0,Y 594.346,Z 241.259,A -85,B 0,C 180,E1 -1106.701,E2 -1106.701} C_VEL
LIN {X 0,Y 594.326,Z 241.263,A -85,B 0,C 180,E1 -1109.779,E2 -1109.779} C_VEL
LIN {X 0,Y 594.328,Z 241.26,A -85,B 0,C 180,E1 -1112.149,E2 -1112.149} C_VEL
LIN {X 0,Y 594.348,Z 241.259,A -85,B 0,C 180,E1 -1114.582,E2 -1114.582} C_VEL
LIN {X 0,Y 594.368,Z 241.258,A -85,B 0,C 180,E1 -1117.607,E2 -1117.607} C_VEL
LIN {X 0,Y 594.333,Z 241.262,A -85,B 0,C 180,E1 -1120.57,E2 -1120.57} C_VEL
LIN {X 0,Y 594.334,Z 241.264,A -85,B 0,C 180,E1 -1123.302,E2 -1123.302} C_VEL
LIN {X 0,Y 594.336,Z 241.259,A -85,B 0,C 180,E1 -1126.164,E2 -1126.164} C_VEL
LIN {X 0,Y 594.351,Z 241.262,A -85,B 0,C 180,E1 -1129.181,E2 -1129.181} C_VEL
LIN {X 0,Y 594.338,Z 241.259,A -85,B 0,C 180,E1 -1132.056,E2 -1132.056} C_VEL
LIN {X 0,Y 594.301,Z 241.272,A -85,B 0,C 180,E1 -1134.683,E2 -1134.683} C_VEL
LIN {X 0,Y 594.334,Z 241.263,A -85,B 0,C 180,E1 -1137.095,E2 -1137.095} C_VEL
LIN {X 0,Y 594.34,Z 241.258,A -85,B 0,C 180,E1 -1139.679,E2 -1139.679} C_VEL
LIN {X 0,Y 594.332,Z 241.269,A -85,B 0,C 180,E1 -1142.538,E2 -1142.538} C_VEL
LIN {X 0,Y 594.323,Z 241.267,A -85,B 0,C 180,E1 -1144.805,E2 -1144.805} C_VEL
LIN {X 0,Y 594.32,Z 241.289,A -85,B 0,C 180,E1 -1147.421,E2 -1147.421} C_VEL
LIN {X 0,Y 594.692,Z 245.893,A -85,B 0,C 180,E1 -1148.145,E2 -1148.145} C_VEL
LIN {X 0,Y 594.561,Z 264.053,A -85,B 0,C 180,E1 -1150.906,E2 -1150.906} C_VEL
LIN {X 0,Y 594.508,Z 281.498,A -85,B 0,C 180,E1 -1153.518,E2 -1153.518} C_VEL
LIN {X 0,Y 594.426,Z 300.488,A -85,B 0,C 180,E1 -1156.323,E2 -1156.323} C_VEL
LIN {X 0,Y 594.326,Z 318.542,A -85,B 0,C 180,E1 -1158.958,E2 -1158.958} C_VEL
LIN {X 0,Y 594.318,Z 322.296,A -85,B 0,C 180,E1 -1159.503,E2 -1159.503} C_VEL
LIN {X 0,Y 594.566,Z 343.219,A -85,B 0,C 180,E1 -1159.766,E2 -1159.766} C_VEL
LIN {X 0,Y 594.472,Z 400.464,A -85,B 0,C 180,E1 -1160.473,E2 -1160.473} C_VEL
LIN {X 0,Y 594.428,Z 410.92,A -85,B 0,C 180,E1 -1160.709,E2 -1160.709} C_VEL
LIN {X 0,Y 594.4,Z 423.542,A -85,B 0,C 180,E1 -1161.159,E2 -1161.159} C_VEL
LIN {X 0,Y 594.422,Z 432.244,A -85,B 0,C 180,E1 -1161.587,E2 -1161.587} C_VEL
LIN {X 0,Y 594.376,Z 440.551,A -85,B 0,C 180,E1 -1162.1,E2 -1162.1} C_VEL
LIN {X 0,Y 594.352,Z 448.406,A -85,B 0,C 180,E1 -1162.697,E2 -1162.697} C_VEL
LIN {X 0,Y 594.342,Z 455.516,A -85,B 0,C 180,E1 -1163.357,E2 -1163.357} C_VEL
LIN {X 0,Y 594.318,Z 463.193,A -85,B 0,C 180,E1 -1164.232,E2 -1164.232} C_VEL
LIN {X 0,Y 594.289,Z 469.03,A -85,B 0,C 180,E1 -1165.082,E2 -1165.082} C_VEL
LIN {X 0,Y 594.261,Z 473.633,A -85,B 0,C 180,E1 -1165.931,E2 -1165.931} C_VEL
LIN {X 0,Y 594.265,Z 476.623,A -85,B 0,C 180,E1 -1166.61,E2 -1166.61} C_VEL
LIN {X 0,Y 594.228,Z 478.934,A -85,B 0,C 180,E1 -1167.289,E2 -1167.289} C_VEL
LIN {X 0,Y 594.242,Z 480.68,A -85,B 0,C 180,E1 -1167.967,E2 -1167.967} C_VEL
LIN {X 0,Y 594.245,Z 481.936,A -85,B 0,C 180,E1 -1168.645,E2 -1168.645} C_VEL
LIN {X 0,Y 594.235,Z 482.713,A -85,B 0,C 180,E1 -1169.323,E2 -1169.323} C_VEL
LIN {X 0,Y 594.233,Z 483,A -85,B 0,C 180,E1 -1170,E2 -1170} C_VEL
LIN {X 0,Y 594.235,Z 482.712,A -85,B 0,C 180,E1 -1170.678,E2 -1170.678} C_VEL
LIN {X 0,Y 594.245,Z 481.935,A -85,B 0,C 180,E1 -1171.356,E2 -1171.356} C_VEL
LIN {X 0,Y 594.242,Z 480.679,A -85,B 0,C 180,E1 -1172.034,E2 -1172.034} C_VEL
LIN {X 0,Y 594.245,Z 477.786,A -85,B 0,C 180,E1 -1173.051,E2 -1173.051} C_VEL
LIN {X 0,Y 594.285,Z 475.145,A -85,B 0,C 180,E1 -1173.73,E2 -1173.73} C_VEL
LIN {X 0,Y 594.256,Z 469.983,A -85,B 0,C 180,E1 -1174.749,E2 -1174.749} C_VEL
LIN {X 0,Y 594.318,Z 463.186,A -85,B 0,C 180,E1 -1175.769,E2 -1175.769} C_VEL
LIN {X 0,Y 594.343,Z 455.512,A -85,B 0,C 180,E1 -1176.644,E2 -1176.644} C_VEL
LIN {X 0,Y 594.353,Z 448.4,A -85,B 0,C 180,E1 -1177.303,E2 -1177.303} C_VEL
LIN {X 0,Y 594.377,Z 440.543,A -85,B 0,C 180,E1 -1177.901,E2 -1177.901} C_VEL
LIN {X 0,Y 594.406,Z 430.731,A -85,B 0,C 180,E1 -1178.499,E2 -1178.499} C_VEL
LIN {X 0,Y 594.422,Z 419.289,A -85,B 0,C 180,E1 -1179.013,E2 -1179.013} C_VEL
LIN {X 0,Y 594.442,Z 409.233,A -85,B 0,C 180,E1 -1179.335,E2 -1179.335} C_VEL
LIN {X 0,Y 594.473,Z 400.425,A -85,B 0,C 180,E1 -1179.527,E2 -1179.527} C_VEL
LIN {X 0,Y 594.459,Z 323.484,A -85,B 0,C 180,E1 -1180.473,E2 -1180.473} C_VEL
LIN {X 0,Y 594.313,Z 322.143,A -85,B 0,C 180,E1 -1180.519,E2 -1180.519} C_VEL
LIN {X 0,Y 594.427,Z 304.043,A -85,B 0,C 180,E1 -1183.156,E2 -1183.156} C_VEL
LIN {X 0,Y 594.49,Z 285.054,A -85,B 0,C 180,E1 -1185.954,E2 -1185.954} C_VEL
LIN {X 0,Y 594.527,Z 267.251,A -85,B 0,C 180,E1 -1188.613,E2 -1188.613} C_VEL
LIN {X 0,Y 594.659,Z 249.296,A -85,B 0,C 180,E1 -1191.334,E2 -1191.334} C_VEL
LIN {X 0,Y 594.635,Z 243.514,A -85,B 0,C 180,E1 -1192.223,E2 -1192.223} C_VEL
LIN {X 0,Y 594.302,Z 241.268,A -85,B 0,C 180,E1 -1192.613,E2 -1192.613} C_VEL
LIN {X 0,Y 594.324,Z 241.267,A -85,B 0,C 180,E1 -1195.196,E2 -1195.196} C_VEL
LIN {X 0,Y 594.343,Z 241.266,A -85,B 0,C 180,E1 -1197.519,E2 -1197.519} C_VEL
LIN {X 0,Y 594.343,Z 241.258,A -85,B 0,C 180,E1 -1200.321,E2 -1200.321} C_VEL
LIN {X 0,Y 594.337,Z 241.263,A -85,B 0,C 180,E1 -1202.953,E2 -1202.953} C_VEL
LIN {X 0,Y 594.298,Z 241.271,A -85,B 0,C 180,E1 -1205.413,E2 -1205.413} C_VEL
LIN {X 0,Y 594.302,Z 241.263,A -85,B 0,C 180,E1 -1207.947,E2 -1207.947} C_VEL
LIN {X 0,Y 594.355,Z 241.262,A -85,B 0,C 180,E1 -1210.819,E2 -1210.819} C_VEL
LIN {X 0,Y 594.332,Z 241.26,A -85,B 0,C 180,E1 -1213.836,E2 -1213.836} C_VEL
LIN {X 0,Y 594.338,Z 241.264,A -85,B 0,C 180,E1 -1216.698,E2 -1216.698} C_VEL
LIN {X 0,Y 594.337,Z 241.261,A -85,B 0,C 180,E1 -1219.43,E2 -1219.43} C_VEL
LIN {X 0,Y 594.353,Z 241.259,A -85,B 0,C 180,E1 -1222.396,E2 -1222.396} C_VEL
LIN {X 0,Y 594.345,Z 241.259,A -85,B 0,C 180,E1 -1225.418,E2 -1225.418} C_VEL
LIN {X 0,Y 594.352,Z 241.261,A -85,B 0,C 180,E1 -1228.362,E2 -1228.362} C_VEL
LIN {X 0,Y 594.337,Z 241.263,A -85,B 0,C 180,E1 -1231.051,E2 -1231.051} C_VEL
LIN {X 0,Y 594.351,Z 241.258,A -85,B 0,C 180,E1 -1233.299,E2 -1233.299} C_VEL
LIN {X 0,Y 594.336,Z 241.264,A -85,B 0,C 180,E1 -1236.294,E2 -1236.294} C_VEL
LIN {X 0,Y 594.367,Z 241.256,A -85,B 0,C 180,E1 -1239.223,E2 -1239.223} C_VEL
LIN {X 0,Y 594.316,Z 241.265,A -85,B 0,C 180,E1 -1242.094,E2 -1242.094} C_VEL
LIN {X 0,Y 594.329,Z 241.262,A -85,B 0,C 180,E1 -1244.921,E2 -1244.921} C_VEL
LIN {X 0,Y 594.34,Z 241.26,A -85,B 0,C 180,E1 -1247.711,E2 -1247.711} C_VEL
LIN {X 0,Y 594.34,Z 241.266,A -85,B 0,C 180,E1 -1250.471,E2 -1250.471} C_VEL
LIN {X 0,Y 594.34,Z 241.258,A -85,B 0,C 180,E1 -1253.209,E2 -1253.209} C_VEL
LIN {X 0,Y 594.346,Z 241.263,A -85,B 0,C 180,E1 -1255.932,E2 -1255.932} C_VEL
LIN {X 0,Y 594.34,Z 241.261,A -85,B 0,C 180,E1 -1258.645,E2 -1258.645} C_VEL
LIN {X 0,Y 594.322,Z 241.263,A -85,B 0,C 180,E1 -1260.678,E2 -1260.678} C_VEL
LIN {X 0,Y 594.365,Z 241.257,A -85,B 0,C 180,E1 -1262.711,E2 -1262.711} C_VEL
LIN {X 0,Y 594.358,Z 241.258,A -85,B 0,C 180,E1 -1265.428,E2 -1265.428} C_VEL
LIN {X 0,Y 594.371,Z 241.261,A -85,B 0,C 180,E1 -1268.157,E2 -1268.157} C_VEL
LIN {X 0,Y 594.331,Z 241.26,A -85,B 0,C 180,E1 -1271.044,E2 -1271.044} C_VEL
LIN {X 0,Y 594.359,Z 241.264,A -85,B 0,C 180,E1 -1273.68,E2 -1273.68} C_VEL
LIN {X 0,Y 594.323,Z 241.263,A -85,B 0,C 180,E1 -1275.283,E2 -1275.283} C_VEL
LIN {X 0,Y 593.653,Z 241.354,A -85,B 0,C 180,E1 -1275.849,E2 -1275.849} C_VEL
LIN {X 0,Y 590.788,Z 241.712,A -85,B 0,C 180,E1 -1276.766,E2 -1276.766} C_VEL
LIN {X 0,Y 588.377,Z 242.01,A -85,B 0,C 180,E1 -1277.505,E2 -1277.505} C_VEL
LIN {X 0,Y 587.353,Z 242.134,A -85,B 0,C 180,E1 -1278.075,E2 -1278.075} C_VEL
LIN {X 0,Y 587.275,Z 242.141,A -85,B 0,C 180,E1 -1278.267,E2 -1278.267} C_VEL
LIN {X 0,Y 587.297,Z 242.137,A -85,B 0,C 180,E1 -1281.039,E2 -1281.039} C_VEL
LIN {X 0,Y 587.284,Z 242.142,A -85,B 0,C 180,E1 -1284.009,E2 -1284.009} C_VEL
LIN {X 0,Y 587.297,Z 242.137,A -85,B 0,C 180,E1 -1286.281,E2 -1286.281} C_VEL
LIN {X 0,Y 587.3,Z 242.139,A -85,B 0,C 180,E1 -1289.124,E2 -1289.124} C_VEL
LIN {X 0,Y 587.315,Z 242.138,A -85,B 0,C 180,E1 -1291.831,E2 -1291.831} C_VEL
LIN {X 0,Y 587.326,Z 242.132,A -85,B 0,C 180,E1 -1294.344,E2 -1294.344} C_VEL
LIN {X 0,Y 587.332,Z 242.137,A -85,B 0,C 180,E1 -1297.609,E2 -1297.609} C_VEL
LIN {X 0,Y 587.292,Z 242.137,A -85,B 0,C 180,E1 -1300.256,E2 -1300.256} C_VEL
LIN {X 0,Y 587.289,Z 242.145,A -85,B 0,C 180,E1 -1303.115,E2 -1303.115} C_VEL
LIN {X 0,Y 587.298,Z 242.136,A -85,B 0,C 180,E1 -1306.047,E2 -1306.047} C_VEL
LIN {X 0,Y 587.308,Z 242.142,A -85,B 0,C 180,E1 -1308.928,E2 -1308.928} C_VEL
LIN {X 0,Y 587.311,Z 242.137,A -85,B 0,C 180,E1 -1311.519,E2 -1311.519} C_VEL
LIN {X 0,Y 587.275,Z 242.139,A -85,B 0,C 180,E1 -1314.099,E2 -1314.099} C_VEL
LIN {X 0,Y 587.332,Z 242.141,A -85,B 0,C 180,E1 -1316.89,E2 -1316.89} C_VEL
LIN {X 0,Y 587.295,Z 242.136,A -85,B 0,C 180,E1 -1319.827,E2 -1319.827} C_VEL
LIN {X 0,Y 587.298,Z 242.138,A -85,B 0,C 180,E1 -1322.317,E2 -1322.317} C_VEL
LIN {X 0,Y 587.299,Z 242.139,A -85,B 0,C 180,E1 -1325.239,E2 -1325.239} C_VEL
LIN {X 0,Y 587.303,Z 242.138,A -85,B 0,C 180,E1 -1328.225,E2 -1328.225} C_VEL
LIN {X 0,Y 587.324,Z 242.135,A -85,B 0,C 180,E1 -1331.15,E2 -1331.15} C_VEL
LIN {X 0,Y 587.318,Z 242.17,A -85,B 0,C 180,E1 -1334.158,E2 -1334.158} C_VEL
LIN {X 0,Y 587.224,Z 253.836,A -85,B 0,C 180,E1 -1336.856,E2 -1336.856} C_VEL
LIN {X 0,Y 587.16,Z 265.192,A -85,B 0,C 180,E1 -1339.455,E2 -1339.455} C_VEL
LIN {X 0,Y 587.578,Z 271.327,A -85,B 0,C 180,E1 -1339.543,E2 -1339.543} C_VEL
LIN {X 0,Y 587.478,Z 340.328,A -85,B 0,C 180,E1 -1340.402,E2 -1340.402} C_VEL
LIN {X 0,Y 587.429,Z 350.004,A -85,B 0,C 180,E1 -1340.618,E2 -1340.618} C_VEL
LIN {X 0,Y 587.385,Z 361.568,A -85,B 0,C 180,E1 -1341.008,E2 -1341.008} C_VEL
LIN {X 0,Y 587.375,Z 371.449,A -85,B 0,C 180,E1 -1341.485,E2 -1341.485} C_VEL
LIN {X 0,Y 587.335,Z 379.904,A -85,B 0,C 180,E1 -1342.004,E2 -1342.004} C_VEL
LIN {X 0,Y 587.295,Z 387.874,A -85,B 0,C 180,E1 -1342.609,E2 -1342.609} C_VEL
LIN {X 0,Y 587.288,Z 394.722,A -85,B 0,C 180,E1 -1343.241,E2 -1343.241} C_VEL
LIN {X 0,Y 587.265,Z 401.406,A -85,B 0,C 180,E1 -1343.989,E2 -1343.989} C_VEL
LIN {X 0,Y 587.172,Z 407.647,A -85,B 0,C 180,E1 -1344.849,E2 -1344.849} C_VEL
LIN {X 0,Y 587.181,Z 413.431,A -85,B 0,C 180,E1 -1345.881,E2 -1345.881} C_VEL
LIN {X 0,Y 587.193,Z 416.446,A -85,B 0,C 180,E1 -1346.569,E2 -1346.569} C_VEL
LIN {X 0,Y 587.135,Z 418.782,A -85,B 0,C 180,E1 -1347.255,E2 -1347.255} C_VEL
LIN {X 0,Y 587.141,Z 420.574,A -85,B 0,C 180,E1 -1347.942,E2 -1347.942} C_VEL
LIN {X 0,Y 587.144,Z 421.873,A -85,B 0,C 180,E1 -1348.628,E2 -1348.628} C_VEL
LIN {X 0,Y 587.136,Z 422.69,A -85,B 0,C 180,E1 -1349.314,E2 -1349.314} C_VEL
LIN {X 0,Y 587.135,Z 422.996,A -85,B 0,C 180,E1 -1350,E2 -1350} C_VEL
LIN {X 0,Y 587.137,Z 422.733,A -85,B 0,C 180,E1 -1350.685,E2 -1350.685} C_VEL
LIN {X 0,Y 587.146,Z 421.998,A -85,B 0,C 180,E1 -1351.371,E2 -1351.371} C_VEL
LIN {X 0,Y 587.142,Z 420.786,A -85,B 0,C 180,E1 -1352.058,E2 -1352.058} C_VEL
LIN {X 0,Y 587.156,Z 417.94,A -85,B 0,C 180,E1 -1353.087,E2 -1353.087} C_VEL
LIN {X 0,Y 587.211,Z 415.348,A -85,B 0,C 180,E1 -1353.774,E2 -1353.774} C_VEL
LIN {X 0,Y 587.17,Z 410.239,A -85,B 0,C 180,E1 -1354.806,E2 -1354.806} C_VEL
LIN {X 0,Y 587.239,Z 404.743,A -85,B 0,C 180,E1 -1355.666,E2 -1355.666} C_VEL
LIN {X 0,Y 587.268,Z 396.749,A -85,B 0,C 180,E1 -1356.643,E2 -1356.643} C_VEL
LIN {X 0,Y 587.296,Z 388.935,A -85,B 0,C 180,E1 -1357.391,E2 -1357.391} C_VEL
LIN {X 0,Y 587.34,Z 381.187,A -85,B 0,C 180,E1 -1357.996,E2 -1357.996} C_VEL
LIN {X 0,Y 587.379,Z 373.02,A -85,B 0,C 180,E1 -1358.515,E2 -1358.515} C_VEL
LIN {X 0,Y 587.382,Z 362.637,A -85,B 0,C 180,E1 -1359.035,E2 -1359.035} C_VEL
LIN {X 0,Y 587.433,Z 350.98,A -85,B 0,C 180,E1 -1359.446,E2 -1359.446} C_VEL
LIN {X 0,Y 587.497,Z 340.56,A -85,B 0,C 180,E1 -1359.684,E2 -1359.684} C_VEL
LIN {X 0,Y 587.593,Z 287.046,A -85,B 0,C 180,E1 -1360.355,E2 -1360.355} C_VEL
LIN {X 0,Y 587.391,Z 266.717,A -85,B 0,C 180,E1 -1360.606,E2 -1360.606} C_VEL
LIN {X 0,Y 587.157,Z 265.144,A -85,B 0,C 180,E1 -1360.646,E2 -1360.646} C_VEL
LIN {X 0,Y 587.204,Z 254.23,A -85,B 0,C 180,E1 -1363.144,E2 -1363.144} C_VEL
LIN {X 0,Y 587.316,Z 242.137,A -85,B 0,C 180,E1 -1365.975,E2 -1365.975} C_VEL
LIN {X 0,Y 587.326,Z 242.136,A -85,B 0,C 180,E1 -1369.034,E2 -1369.034} C_VEL
LIN {X 0,Y 587.293,Z 242.14,A -85,B 0,C 180,E1 -1371.775,E2 -1371.775} C_VEL
LIN {X 0,Y 587.295,Z 242.138,A -85,B 0,C 180,E1 -1374.761,E2 -1374.761} C_VEL
LIN {X 0,Y 587.293,Z 242.14,A -85,B 0,C 180,E1 -1377.682,E2 -1377.682} C_VEL
LIN {X 0,Y 587.302,Z 242.136,A -85,B 0,C 180,E1 -1380.504,E2 -1380.504} C_VEL
LIN {X 0,Y 587.315,Z 242.139,A -85,B 0,C 180,E1 -1383.397,E2 -1383.397} C_VEL
LIN {X 0,Y 587.261,Z 242.141,A -85,B 0,C 180,E1 -1385.902,E2 -1385.902} C_VEL
LIN {X 0,Y 587.306,Z 242.137,A -85,B 0,C 180,E1 -1388.481,E2 -1388.481} C_VEL
LIN {X 0,Y 587.304,Z 242.142,A -85,B 0,C 180,E1 -1391.159,E2 -1391.159} C_VEL
LIN {X 0,Y 587.298,Z 242.136,A -85,B 0,C 180,E1 -1394.11,E2 -1394.11} C_VEL
LIN {X 0,Y 587.281,Z 242.146,A -85,B 0,C 180,E1 -1396.99,E2 -1396.99} C_VEL
LIN {X 0,Y 587.287,Z 242.137,A -85,B 0,C 180,E1 -1399.743,E2 -1399.743} C_VEL
LIN {X 0,Y 587.326,Z 242.137,A -85,B 0,C 180,E1 -1402.391,E2 -1402.391} C_VEL
LIN {X 0,Y 587.315,Z 242.134,A -85,B 0,C 180,E1 -1405.656,E2 -1405.656} C_VEL
LIN {X 0,Y 587.327,Z 242.137,A -85,B 0,C 180,E1 -1408.23,E2 -1408.23} C_VEL
LIN {X 0,Y 587.294,Z 242.141,A -85,B 0,C 180,E1 -1410.875,E2 -1410.875} C_VEL
LIN {X 0,Y 587.297,Z 242.137,A -85,B 0,C 180,E1 -1413.83,E2 -1413.83} C_VEL
LIN {X 0,Y 587.282,Z 242.143,A -85,B 0,C 180,E1 -1416.74,E2 -1416.74} C_VEL
LIN {X 0,Y 587.294,Z 242.138,A -85,B 0,C 180,E1 -1419.694,E2 -1419.694} C_VEL
LIN {X 0,Y 587.268,Z 242.143,A -85,B 0,C 180,E1 -1421.871,E2 -1421.871} C_VEL
LIN {X 0,Y 587.29,Z 242.14,A -85,B 0,C 180,E1 -1424.736,E2 -1424.736} C_VEL
LIN {X 0,Y 587.265,Z 242.141,A -85,B 0,C 180,E1 -1426.857,E2 -1426.857} C_VEL
LIN {X 0,Y 587.313,Z 242.137,A -85,B 0,C 180,E1 -1429.66,E2 -1429.66} C_VEL
LIN {X 0,Y 587.304,Z 242.14,A -85,B 0,C 180,E1 -1432.436,E2 -1432.436} C_VEL
LIN {X 0,Y 587.317,Z 242.134,A -85,B 0,C 180,E1 -1435.195,E2 -1435.195} C_VEL
LIN {X 0,Y 587.367,Z 242.137,A -85,B 0,C 180,E1 -1437.943,E2 -1437.943} C_VEL
LIN {X 0,Y 587.375,Z 242.135,A -85,B 0,C 180,E1 -1440,E2 -1440} C_VEL
LIN {X 0,Y 587.326,Z 242.132,A -85,B 0,C 180,E1 -1442.743,E2 -1442.743} C_VEL
LIN {X 0,Y 587.326,Z 242.137,A -85,B 0,C 180,E1 -1445.493,E2 -1445.493} C_VEL
LIN {X 0,Y 587.32,Z 242.136,A -85,B 0,C 180,E1 -1448.256,E2 -1448.256} C_VEL
LIN {X 0,Y 587.309,Z 242.136,A -85,B 0,C 180,E1 -1451.117,E2 -1451.117} C_VEL
LIN {X 0,Y 587.311,Z 242.136,A -85,B 0,C 180,E1 -1454.241,E2 -1454.241} C_VEL
LIN {X 0,Y 587.286,Z 242.138,A -85,B 0,C 180,E1 -1456.795,E2 -1456.795} C_VEL
LIN {X 0,Y 587.288,Z 242.146,A -85,B 0,C 180,E1 -1459.577,E2 -1459.577} C_VEL
LIN {X 0,Y 587.287,Z 242.142,A -85,B 0,C 180,E1 -1461.776,E2 -1461.776} C_VEL
LIN {X 0,Y 587.29,Z 242.138,A -85,B 0,C 180,E1 -1464.761,E2 -1464.761} C_VEL
LIN {X 0,Y 587.289,Z 242.141,A -85,B 0,C 180,E1 -1467.682,E2 -1467.682} C_VEL
LIN {X 0,Y 587.281,Z 242.138,A -85,B 0,C 180,E1 -1470.502,E2 -1470.502} C_VEL
LIN {X 0,Y 587.311,Z 242.141,A -85,B 0,C 180,E1 -1473.398,E2 -1473.398} C_VEL
LIN {X 0,Y 587.255,Z 242.142,A -85,B 0,C 180,E1 -1475.903,E2 -1475.903} C_VEL
LIN {X 0,Y 587.293,Z 242.138,A -85,B 0,C 180,E1 -1478.482,E2 -1478.482} C_VEL
LIN {X 0,Y 587.3,Z 242.144,A -85,B 0,C 180,E1 -1481.16,E2 -1481.16} C_VEL
LIN {X 0,Y 587.296,Z 242.136,A -85,B 0,C 180,E1 -1484.111,E2 -1484.111} C_VEL
LIN {X 0,Y 587.276,Z 242.148,A -85,B 0,C 180,E1 -1486.991,E2 -1486.991} C_VEL
LIN {X 0,Y 587.285,Z 242.137,A -85,B 0,C 180,E1 -1489.744,E2 -1489.744} C_VEL
LIN {X 0,Y 587.324,Z 242.136,A -85,B 0,C 180,E1 -1492.391,E2 -1492.391} C_VEL
LIN {X 0,Y 587.294,Z 242.136,A -85,B 0,C 180,E1 -1495.776,E2 -1495.776} C_VEL
LIN {X 0,Y 587.294,Z 242.139,A -85,B 0,C 180,E1 -1498.229,E2 -1498.229} C_VEL
LIN {X 0,Y 587.292,Z 242.143,A -85,B 0,C 180,E1 -1500.877,E2 -1500.877} C_VEL
LIN {X 0,Y 587.29,Z 242.138,A -85,B 0,C 180,E1 -1503.833,E2 -1503.833} C_VEL
LIN {X 0,Y 587.279,Z 242.147,A -85,B 0,C 180,E1 -1506.74,E2 -1506.74} C_VEL
LIN {X 0,Y 587.297,Z 242.287,A -85,B 0,C 180,E1 -1507.292,E2 -1507.292} C_VEL
LIN {X 0,Y 587.76,Z 247.079,A -85,B 0,C 180,E1 -1508.059,E2 -1508.059} C_VEL
LIN {X 0,Y 587.605,Z 264.394,A -85,B 0,C 180,E1 -1510.723,E2 -1510.723} C_VEL
LIN {X 0,Y 587.5,Z 281.498,A -85,B 0,C 180,E1 -1513.316,E2 -1513.316} C_VEL
LIN {X 0,Y 587.418,Z 300.488,A -85,B 0,C 180,E1 -1516.156,E2 -1516.156} C_VEL
LIN {X 0,Y 587.289,Z 319.477,A -85,B 0,C 180,E1 -1518.962,E2 -1518.962} C_VEL
LIN {X 0,Y 587.257,Z 322.344,A -85,B 0,C 180,E1 -1519.383,E2 -1519.383} C_VEL
LIN {X 0,Y 587.551,Z 331.058,A -85,B 0,C 180,E1 -1519.494,E2 -1519.494} C_VEL
LIN {X 0,Y 587.514,Z 399.164,A -85,B 0,C 180,E1 -1520.338,E2 -1520.338} C_VEL
LIN {X 0,Y 587.452,Z 408.429,A -85,B 0,C 180,E1 -1520.532,E2 -1520.532} C_VEL
LIN {X 0,Y 587.415,Z 416.903,A -85,B 0,C 180,E1 -1520.792,E2 -1520.792} C_VEL
LIN {X 0,Y 587.365,Z 425.407,A -85,B 0,C 180,E1 -1521.139,E2 -1521.139} C_VEL
LIN {X 0,Y 587.39,Z 433.735,A -85,B 0,C 180,E1 -1521.572,E2 -1521.572} C_VEL
LIN {X 0,Y 587.334,Z 441.771,A -85,B 0,C 180,E1 -1522.091,E2 -1522.091} C_VEL
LIN {X 0,Y 587.29,Z 449.421,A -85,B 0,C 180,E1 -1522.696,E2 -1522.696} C_VEL
LIN {X 0,Y 587.281,Z 457.809,A -85,B 0,C 180,E1 -1523.512,E2 -1523.512} C_VEL
LIN {X 0,Y 587.238,Z 464.435,A -85,B 0,C 180,E1 -1524.334,E2 -1524.334} C_VEL
LIN {X 0,Y 587.17,Z 469.989,A -85,B 0,C 180,E1 -1525.194,E2 -1525.194} C_VEL
LIN {X 0,Y 587.21,Z 475.149,A -85,B 0,C 180,E1 -1526.226,E2 -1526.226} C_VEL
LIN {X 0,Y 587.155,Z 477.789,A -85,B 0,C 180,E1 -1526.913,E2 -1526.913} C_VEL
LIN {X 0,Y 587.141,Z 480.681,A -85,B 0,C 180,E1 -1527.942,E2 -1527.942} C_VEL
LIN {X 0,Y 587.145,Z 481.936,A -85,B 0,C 180,E1 -1528.629,E2 -1528.629} C_VEL
LIN {X 0,Y 587.136,Z 482.712,A -85,B 0,C 180,E1 -1529.315,E2 -1529.315} C_VEL
LIN {X 0,Y 587.134,Z 483,A -85,B 0,C 180,E1 -1530,E2 -1530} C_VEL
LIN {X 0,Y 587.136,Z 482.711,A -85,B 0,C 180,E1 -1530.686,E2 -1530.686} C_VEL
LIN {X 0,Y 587.145,Z 481.935,A -85,B 0,C 180,E1 -1531.372,E2 -1531.372} C_VEL
LIN {X 0,Y 587.141,Z 480.679,A -85,B 0,C 180,E1 -1532.058,E2 -1532.058} C_VEL
LIN {X 0,Y 587.155,Z 477.787,A -85,B 0,C 180,E1 -1533.088,E2 -1533.088} C_VEL
LIN {X 0,Y 587.21,Z 475.146,A -85,B 0,C 180,E1 -1533.775,E2 -1533.775} C_VEL
LIN {X 0,Y 587.17,Z 469.983,A -85,B 0,C 180,E1 -1534.806,E2 -1534.806} C_VEL
LIN {X 0,Y 587.253,Z 463.185,A -85,B 0,C 180,E1 -1535.839,E2 -1535.839} C_VEL
LIN {X 0,Y 587.269,Z 456.284,A -85,B 0,C 180,E1 -1536.646,E2 -1536.646} C_VEL
LIN {X 0,Y 587.295,Z 448.402,A -85,B 0,C 180,E1 -1537.391,E2 -1537.391} C_VEL
LIN {X 0,Y 587.339,Z 440.545,A -85,B 0,C 180,E1 -1537.996,E2 -1537.996} C_VEL
LIN {X 0,Y 587.379,Z 430.729,A -85,B 0,C 180,E1 -1538.602,E2 -1538.602} C_VEL
LIN {X 0,Y 587.419,Z 419.291,A -85,B 0,C 180,E1 -1539.122,E2 -1539.122} C_VEL
LIN {X 0,Y 587.45,Z 409.233,A -85,B 0,C 180,E1 -1539.447,E2 -1539.447} C_VEL
LIN {X 0,Y 587.484,Z 400.425,A -85,B 0,C 180,E1 -1539.642,E2 -1539.642} C_VEL
LIN {X 0,Y 587.499,Z 324.042,A -85,B 0,C 180,E1 -1540.592,E2 -1540.592} C_VEL
LIN {X 0,Y 587.264,Z 322.197,A -85,B 0,C 180,E1 -1540.639,E2 -1540.639} C_VEL
LIN {X 0,Y 587.409,Z 304.043,A -85,B 0,C 180,E1 -1543.316,E2 -1543.316} C_VEL
LIN {X 0,Y 587.487,Z 283.867,A -85,B 0,C 180,E1 -1546.328,E2 -1546.328} C_VEL
LIN {X 0,Y 587.57,Z 267.251,A -85,B 0,C 180,E1 -1548.842,E2 -1548.842} C_VEL
LIN {X 0,Y 587.721,Z 250.637,A -85,B 0,C 180,E1 -1551.39,E2 -1551.39} C_VEL
LIN {X 0,Y 587.529,Z 243.514,A -85,B 0,C 180,E1 -1552.506,E2 -1552.506} C_VEL
LIN {X 0,Y 587.283,Z 242.143,A -85,B 0,C 180,E1 -1552.732,E2 -1552.732} C_VEL
LIN {X 0,Y 587.294,Z 242.145,A -85,B 0,C 180,E1 -1555.519,E2 -1555.519} C_VEL
LIN {X 0,Y 587.283,Z 242.141,A -85,B 0,C 180,E1 -1557.821,E2 -1557.821} C_VEL
LIN {X 0,Y 587.284,Z 242.137,A -85,B 0,C 180,E1 -1560.501,E2 -1560.501} C_VEL
LIN {X 0,Y 587.299,Z 242.143,A -85,B 0,C 180,E1 -1563.399,E2 -1563.399} C_VEL
LIN {X 0,Y 587.251,Z 242.142,A -85,B 0,C 180,E1 -1565.903,E2 -1565.903} C_VEL
LIN {X 0,Y 587.27,Z 242.14,A -85,B 0,C 180,E1 -1568.484,E2 -1568.484} C_VEL
LIN {X 0,Y 587.297,Z 242.145,A -85,B 0,C 180,E1 -1571.161,E2 -1571.161} C_VEL
LIN {X 0,Y 587.287,Z 242.137,A -85,B 0,C 180,E1 -1574.109,E2 -1574.109} C_VEL
LIN {X 0,Y 587.28,Z 242.148,A -85,B 0,C 180,E1 -1576.99,E2 -1576.99} C_VEL
LIN {X 0,Y 587.289,Z 242.137,A -85,B 0,C 180,E1 -1579.744,E2 -1579.744} C_VEL
LIN {X 0,Y 587.307,Z 242.137,A -85,B 0,C 180,E1 -1582.39,E2 -1582.39} C_VEL
LIN {X 0,Y 587.307,Z 242.135,A -85,B 0,C 180,E1 -1585.658,E2 -1585.658} C_VEL
LIN {X 0,Y 587.298,Z 242.138,A -85,B 0,C 180,E1 -1588.229,E2 -1588.229} C_VEL
LIN {X 0,Y 587.296,Z 242.143,A -85,B 0,C 180,E1 -1590.876,E2 -1590.876} C_VEL
LIN {X 0,Y 587.294,Z 242.137,A -85,B 0,C 180,E1 -1593.832,E2 -1593.832} C_VEL
LIN {X 0,Y 587.284,Z 242.145,A -85,B 0,C 180,E1 -1596.74,E2 -1596.74} C_VEL
LIN {X 0,Y 587.295,Z 242.136,A -85,B 0,C 180,E1 -1599.694,E2 -1599.694} C_VEL
LIN {X 0,Y 587.269,Z 242.148,A -85,B 0,C 180,E1 -1602.592,E2 -1602.592} C_VEL
LIN {X 0,Y 587.303,Z 242.135,A -85,B 0,C 180,E1 -1605.446,E2 -1605.446} C_VEL
LIN {X 0,Y 587.311,Z 242.143,A -85,B 0,C 180,E1 -1608.263,E2 -1608.263} C_VEL
LIN {X 0,Y 587.275,Z 242.139,A -85,B 0,C 180,E1 -1611.05,E2 -1611.05} C_VEL
LIN {X 0,Y 587.304,Z 242.139,A -85,B 0,C 180,E1 -1613.817,E2 -1613.817} C_VEL
LIN {X 0,Y 587.298,Z 242.141,A -85,B 0,C 180,E1 -1615.883,E2 -1615.883} C_VEL
LIN {X 0,Y 587.3,Z 242.138,A -85,B 0,C 180,E1 -1618.629,E2 -1618.629} C_VEL
LIN {X 0,Y 587.277,Z 242.14,A -85,B 0,C 180,E1 -1620.686,E2 -1620.686} C_VEL
LIN {X 0,Y 587.333,Z 242.132,A -85,B 0,C 180,E1 -1622.744,E2 -1622.744} C_VEL
LIN {X 0,Y 587.327,Z 242.135,A -85,B 0,C 180,E1 -1625.493,E2 -1625.493} C_VEL
LIN {X 0,Y 587.327,Z 242.137,A -85,B 0,C 180,E1 -1628.256,E2 -1628.256} C_VEL
LIN {X 0,Y 587.298,Z 242.136,A -85,B 0,C 180,E1 -1631.107,E2 -1631.107} C_VEL
LIN {X 0,Y 587.335,Z 242.141,A -85,B 0,C 180,E1 -1633.846,E2 -1633.846} C_VEL
LIN {X 0,Y 587.293,Z 242.136,A -85,B 0,C 180,E1 -1636.795,E2 -1636.795} C_VEL
LIN {X 0,Y 587.275,Z 242.141,A -85,B 0,C 180,E1 -1638.267,E2 -1638.267} C_VEL
LIN {X 0,Y 586.622,Z 242.222,A -85,B 0,C 180,E1 -1638.84,E2 -1638.84} C_VEL
LIN {X 0,Y 583.767,Z 242.585,A -85,B 0,C 180,E1 -1639.768,E2 -1639.768} C_VEL
LIN {X 0,Y 581.358,Z 242.88,A -85,B 0,C 180,E1 -1640.515,E2 -1640.515} C_VEL
LIN {X 0,Y 580.339,Z 243.005,A -85,B 0,C 180,E1 -1641.092,E2 -1641.092} C_VEL
LIN {X 0,Y 580.265,Z 243.016,A -85,B 0,C 180,E1 -1641.287,E2 -1641.287} C_VEL
LIN {X 0,Y 580.248,Z 243.015,A -85,B 0,C 180,E1 -1644.319,E2 -1644.319} C_VEL
LIN {X 0,Y 580.24,Z 243.015,A -85,B 0,C 180,E1 -1646.625,E2 -1646.625} C_VEL
LIN {X 0,Y 580.25,Z 243.021,A -85,B 0,C 180,E1 -1649.3,E2 -1649.3} C_VEL
LIN {X 0,Y 580.283,Z 243.011,A -85,B 0,C 180,E1 -1652.202,E2 -1652.202} C_VEL
LIN {X 0,Y 580.273,Z 243.012,A -85,B 0,C 180,E1 -1654.698,E2 -1654.698} C_VEL
LIN {X 0,Y 580.282,Z 243.019,A -85,B 0,C 180,E1 -1657.27,E2 -1657.27} C_VEL
LIN {X 0,Y 580.274,Z 243.011,A -85,B 0,C 180,E1 -1660.268,E2 -1660.268} C_VEL
LIN {X 0,Y 580.251,Z 243.016,A -85,B 0,C 180,E1 -1662.709,E2 -1662.709} C_VEL
LIN {X 0,Y 580.251,Z 243.017,A -85,B 0,C 180,E1 -1665.611,E2 -1665.611} C_VEL
LIN {X 0,Y 580.239,Z 243.015,A -85,B 0,C 180,E1 -1668.227,E2 -1668.227} C_VEL
LIN {X 0,Y 580.264,Z 243.021,A -85,B 0,C 180,E1 -1670.964,E2 -1670.964} C_VEL
LIN {X 0,Y 580.244,Z 243.017,A -85,B 0,C 180,E1 -1673.594,E2 -1673.594} C_VEL
LIN {X 0,Y 580.271,Z 243.012,A -85,B 0,C 180,E1 -1676.142,E2 -1676.142} C_VEL
LIN {X 0,Y 580.253,Z 243.019,A -85,B 0,C 180,E1 -1678.613,E2 -1678.613} C_VEL
LIN {X 0,Y 580.276,Z 243.018,A -85,B 0,C 180,E1 -1681.023,E2 -1681.023} C_VEL
LIN {X 0,Y 580.262,Z 243.013,A -85,B 0,C 180,E1 -1683.672,E2 -1683.672} C_VEL
LIN {X 0,Y 580.246,Z 243.019,A -85,B 0,C 180,E1 -1686.44,E2 -1686.44} C_VEL
LIN {X 0,Y 580.252,Z 243.014,A -85,B 0,C 180,E1 -1689.436,E2 -1689.436} C_VEL
LIN {X 0,Y 580.238,Z 243.015,A -85,B 0,C 180,E1 -1691.644,E2 -1691.644} C_VEL
LIN {X 0,Y 580.267,Z 243.128,A -85,B 0,C 180,E1 -1694.186,E2 -1694.186} C_VEL
LIN {X 0,Y 580.167,Z 255.369,A -85,B 0,C 180,E1 -1697.049,E2 -1697.049} C_VEL
LIN {X 0,Y 580.097,Z 265.164,A -85,B 0,C 180,E1 -1699.318,E2 -1699.318} C_VEL
LIN {X 0,Y 580.619,Z 269.889,A -85,B 0,C 180,E1 -1699.398,E2 -1699.398} C_VEL
LIN {X 0,Y 580.496,Z 340.359,A -85,B 0,C 180,E1 -1700.285,E2 -1700.285} C_VEL
LIN {X 0,Y 580.422,Z 350.025,A -85,B 0,C 180,E1 -1700.504,E2 -1700.504} C_VEL
LIN {X 0,Y 580.377,Z 361.58,A -85,B 0,C 180,E1 -1700.898,E2 -1700.898} C_VEL
LIN {X 0,Y 580.359,Z 371.456,A -85,B 0,C 180,E1 -1701.381,E2 -1701.381} C_VEL
LIN {X 0,Y 580.294,Z 379.909,A -85,B 0,C 180,E1 -1701.906,E2 -1701.906} C_VEL
LIN {X 0,Y 580.254,Z 387.878,A -85,B 0,C 180,E1 -1702.518,E2 -1702.518} C_VEL
LIN {X 0,Y 580.229,Z 395.027,A -85,B 0,C 180,E1 -1703.189,E2 -1703.189} C_VEL
LIN {X 0,Y 580.209,Z 401.409,A -85,B 0,C 180,E1 -1703.916,E2 -1703.916} C_VEL
LIN {X 0,Y 580.091,Z 407.65,A -85,B 0,C 180,E1 -1704.786,E2 -1704.786} C_VEL
LIN {X 0,Y 580.104,Z 413.434,A -85,B 0,C 180,E1 -1705.831,E2 -1705.831} C_VEL
LIN {X 0,Y 580.122,Z 416.448,A -85,B 0,C 180,E1 -1706.527,E2 -1706.527} C_VEL
LIN {X 0,Y 580.046,Z 418.784,A -85,B 0,C 180,E1 -1707.222,E2 -1707.222} C_VEL
LIN {X 0,Y 580.041,Z 420.576,A -85,B 0,C 180,E1 -1707.917,E2 -1707.917} C_VEL
LIN {X 0,Y 580.044,Z 421.872,A -85,B 0,C 180,E1 -1708.611,E2 -1708.611} C_VEL
LIN {X 0,Y 580.036,Z 422.689,A -85,B 0,C 180,E1 -1709.305,E2 -1709.305} C_VEL
LIN {X 0,Y 580.036,Z 422.996,A -85,B 0,C 180,E1 -1710,E2 -1710} C_VEL
LIN {X 0,Y 580.037,Z 422.731,A -85,B 0,C 180,E1 -1710.694,E2 -1710.694} C_VEL
LIN {X 0,Y 580.046,Z 421.998,A -85,B 0,C 180,E1 -1711.388,E2 -1711.388} C_VEL
LIN {X 0,Y 580.041,Z 420.786,A -85,B 0,C 180,E1 -1712.083,E2 -1712.083} C_VEL
LIN {X 0,Y 580.071,Z 417.939,A -85,B 0,C 180,E1 -1713.125,E2 -1713.125} C_VEL
LIN {X 0,Y 580.123,Z 415.346,A -85,B 0,C 180,E1 -1713.82,E2 -1713.82} C_VEL
LIN {X 0,Y 580.075,Z 410.237,A -85,B 0,C 180,E1 -1714.865,E2 -1714.865} C_VEL
LIN {X 0,Y 580.174,Z 404.74,A -85,B 0,C 180,E1 -1715.735,E2 -1715.735} C_VEL
LIN {X 0,Y 580.195,Z 397.507,A -85,B 0,C 180,E1 -1716.645,E2 -1716.645} C_VEL
LIN {X 0,Y 580.254,Z 388.929,A -85,B 0,C 180,E1 -1717.481,E2 -1717.481} C_VEL
LIN {X 0,Y 580.325,Z 381.18,A -85,B 0,C 180,E1 -1718.093,E2 -1718.093} C_VEL
LIN {X 0,Y 580.36,Z 373.008,A -85,B 0,C 180,E1 -1718.618,E2 -1718.618} C_VEL
LIN {X 0,Y 580.38,Z 362.622,A -85,B 0,C 180,E1 -1719.145,E2 -1719.145} C_VEL
LIN {X 0,Y 580.422,Z 350.959,A -85,B 0,C 180,E1 -1719.561,E2 -1719.561} C_VEL
LIN {X 0,Y 580.52,Z 340.525,A -85,B 0,C 180,E1 -1719.802,E2 -1719.802} C_VEL
LIN {X 0,Y 580.585,Z 288.66,A -85,B 0,C 180,E1 -1720.461,E2 -1720.461} C_VEL
LIN {X 0,Y 580.436,Z 267.688,A -85,B 0,C 180,E1 -1720.722,E2 -1720.722} C_VEL
LIN {X 0,Y 580.088,Z 265.129,A -85,B 0,C 180,E1 -1720.78,E2 -1720.78} C_VEL
LIN {X 0,Y 580.161,Z 254.228,A -85,B 0,C 180,E1 -1723.306,E2 -1723.306} C_VEL
LIN {X 0,Y 580.251,Z 243.018,A -85,B 0,C 180,E1 -1725.949,E2 -1725.949} C_VEL
LIN {X 0,Y 580.297,Z 243.014,A -85,B 0,C 180,E1 -1729.15,E2 -1729.15} C_VEL
LIN {X 0,Y 580.228,Z 243.018,A -85,B 0,C 180,E1 -1732.054,E2 -1732.054} C_VEL
LIN {X 0,Y 580.271,Z 243.018,A -85,B 0,C 180,E1 -1735.081,E2 -1735.081} C_VEL
LIN {X 0,Y 580.238,Z 243.017,A -85,B 0,C 180,E1 -1737.847,E2 -1737.847} C_VEL
LIN {X 0,Y 580.253,Z 243.016,A -85,B 0,C 180,E1 -1740.689,E2 -1740.689} C_VEL
LIN {X 0,Y 580.273,Z 243.018,A -85,B 0,C 180,E1 -1743.311,E2 -1743.311} C_VEL
LIN {X 0,Y 580.212,Z 243.02,A -85,B 0,C 180,E1 -1745.751,E2 -1745.751} C_VEL
LIN {X 0,Y 580.275,Z 243.011,A -85,B 0,C 180,E1 -1748.147,E2 -1748.147} C_VEL
LIN {X 0,Y 580.271,Z 243.02,A -85,B 0,C 180,E1 -1750.845,E2 -1750.845} C_VEL
LIN {X 0,Y 580.231,Z 243.017,A -85,B 0,C 180,E1 -1753.662,E2 -1753.662} C_VEL
LIN {X 0,Y 580.232,Z 243.019,A -85,B 0,C 180,E1 -1756.338,E2 -1756.338} C_VEL
LIN {X 0,Y 580.251,Z 243.018,A -85,B 0,C 180,E1 -1759.152,E2 -1759.152} C_VEL
LIN {X 0,Y 580.271,Z 243.012,A -85,B 0,C 180,E1 -1761.929,E2 -1761.929} C_VEL
LIN {X 0,Y 580.218,Z 243.024,A -85,B 0,C 180,E1 -1764.45,E2 -1764.45} C_VEL
LIN {X 0,Y 580.275,Z 243.015,A -85,B 0,C 180,E1 -1766.974,E2 -1766.974} C_VEL
LIN {X 0,Y 580.262,Z 243.013,A -85,B 0,C 180,E1 -1769.423,E2 -1769.423} C_VEL
LIN {X 0,Y 580.234,Z 243.02,A -85,B 0,C 180,E1 -1772.152,E2 -1772.152} C_VEL
LIN {X 0,Y 580.274,Z 243.014,A -85,B 0,C 180,E1 -1774.919,E2 -1774.919} C_VEL
LIN {X 0,Y 580.225,Z 243.02,A -85,B 0,C 180,E1 -1777.945,E2 -1777.945} C_VEL
LIN {X 0,Y 580.269,Z 243.013,A -85,B 0,C 180,E1 -1780.912,E2 -1780.912} C_VEL
LIN {X 0,Y 580.229,Z 243.02,A -85,B 0,C 180,E1 -1783.824,E2 -1783.824} C_VEL
LIN {X 0,Y 580.287,Z 243.015,A -85,B 0,C 180,E1 -1785.982,E2 -1785.982} C_VEL
LIN {X 0,Y 580.261,Z 243.014,A -85,B 0,C 180,E1 -1788.826,E2 -1788.826} C_VEL
LIN {X 0,Y 580.288,Z 243.012,A -85,B 0,C 180,E1 -1791.643,E2 -1791.643} C_VEL
LIN {X 0,Y 580.298,Z 243.012,A -85,B 0,C 180,E1 -1794.44,E2 -1794.44} C_VEL
LIN {X 0,Y 580.336,Z 243.012,A -85,B 0,C 180,E1 -1797.918,E2 -1797.918} C_VEL
LIN {X 0,Y 580.343,Z 243.011,A -85,B 0,C 180,E1 -1800,E2 -1800} C_VEL
LIN {X 0,Y 580.294,Z 243.008,A -85,B 0,C 180,E1 -1802.777,E2 -1802.777} C_VEL
LIN {X 0,Y 580.295,Z 243.014,A -85,B 0,C 180,E1 -1805.56,E2 -1805.56} C_VEL
LIN {X 0,Y 580.286,Z 243.011,A -85,B 0,C 180,E1 -1808.357,E2 -1808.357} C_VEL
LIN {X 0,Y 580.261,Z 243.015,A -85,B 0,C 180,E1 -1811.174,E2 -1811.174} C_VEL
LIN {X 0,Y 580.285,Z 243.013,A -85,B 0,C 180,E1 -1814.018,E2 -1814.018} C_VEL
LIN {X 0,Y 580.244,Z 243.016,A -85,B 0,C 180,E1 -1816.899,E2 -1816.899} C_VEL
LIN {X 0,Y 580.262,Z 243.017,A -85,B 0,C 180,E1 -1819.824,E2 -1819.824} C_VEL
LIN {X 0,Y 580.221,Z 243.019,A -85,B 0,C 180,E1 -1822.055,E2 -1822.055} C_VEL
LIN {X 0,Y 580.243,Z 243.016,A -85,B 0,C 180,E1 -1824.715,E2 -1824.715} C_VEL
LIN {X 0,Y 580.238,Z 243.025,A -85,B 0,C 180,E1 -1827.404,E2 -1827.404} C_VEL
LIN {X 0,Y 580.239,Z 243.018,A -85,B 0,C 180,E1 -1829.775,E2 -1829.775} C_VEL
LIN {X 0,Y 580.275,Z 243.011,A -85,B 0,C 180,E1 -1832.202,E2 -1832.202} C_VEL
LIN {X 0,Y 580.263,Z 243.015,A -85,B 0,C 180,E1 -1834.698,E2 -1834.698} C_VEL
LIN {X 0,Y 580.273,Z 243.019,A -85,B 0,C 180,E1 -1837.27,E2 -1837.27} C_VEL
LIN {X 0,Y 580.266,Z 243.012,A -85,B 0,C 180,E1 -1840.268,E2 -1840.268} C_VEL
LIN {X 0,Y 580.241,Z 243.02,A -85,B 0,C 180,E1 -1842.71,E2 -1842.71} C_VEL
LIN {X 0,Y 580.245,Z 243.016,A -85,B 0,C 180,E1 -1845.612,E2 -1845.612} C_VEL
LIN {X 0,Y 580.233,Z 243.017,A -85,B 0,C 180,E1 -1848.228,E2 -1848.228} C_VEL
LIN {X 0,Y 580.253,Z 243.021,A -85,B 0,C 180,E1 -1850.964,E2 -1850.964} C_VEL
LIN {X 0,Y 580.226,Z 243.017,A -85,B 0,C 180,E1 -1853.594,E2 -1853.594} C_VEL
LIN {X 0,Y 580.249,Z 243.015,A -85,B 0,C 180,E1 -1856.141,E2 -1856.141} C_VEL
LIN {X 0,Y 580.233,Z 243.024,A -85,B 0,C 180,E1 -1858.613,E2 -1858.613} C_VEL
LIN {X 0,Y 580.238,Z 243.019,A -85,B 0,C 180,E1 -1861.021,E2 -1861.021} C_VEL
LIN {X 0,Y 580.244,Z 243.015,A -85,B 0,C 180,E1 -1863.676,E2 -1863.676} C_VEL
LIN {X 0,Y 580.234,Z 243.025,A -85,B 0,C 180,E1 -1866.441,E2 -1866.441} C_VEL
LIN {X 0,Y 580.263,Z 243.219,A -85,B 0,C 180,E1 -1867.197,E2 -1867.197} C_VEL
LIN {X 0,Y 580.802,Z 248.146,A -85,B 0,C 180,E1 -1867.969,E2 -1867.969} C_VEL
LIN {X 0,Y 580.629,Z 266.158,A -85,B 0,C 180,E1 -1870.755,E2 -1870.755} C_VEL
LIN {X 0,Y 580.518,Z 282.685,A -85,B 0,C 180,E1 -1873.29,E2 -1873.29} C_VEL
LIN {X 0,Y 580.393,Z 301.674,A -85,B 0,C 180,E1 -1876.164,E2 -1876.164} C_VEL
LIN {X 0,Y 580.238,Z 320.556,A -85,B 0,C 180,E1 -1878.987,E2 -1878.987} C_VEL
LIN {X 0,Y 580.198,Z 322.281,A -85,B 0,C 180,E1 -1879.243,E2 -1879.243} C_VEL
LIN {X 0,Y 580.614,Z 329.39,A -85,B 0,C 180,E1 -1879.347,E2 -1879.347} C_VEL
LIN {X 0,Y 580.538,Z 399.163,A -85,B 0,C 180,E1 -1880.221,E2 -1880.221} C_VEL
LIN {X 0,Y 580.466,Z 408.429,A -85,B 0,C 180,E1 -1880.417,E2 -1880.417} C_VEL
LIN {X 0,Y 580.422,Z 416.903,A -85,B 0,C 180,E1 -1880.68,E2 -1880.68} C_VEL
LIN {X 0,Y 580.35,Z 425.409,A -85,B 0,C 180,E1 -1881.031,E2 -1881.031} C_VEL
LIN {X 0,Y 580.346,Z 433.738,A -85,B 0,C 180,E1 -1881.469,E2 -1881.469} C_VEL
LIN {X 0,Y 580.308,Z 441.773,A -85,B 0,C 180,E1 -1881.995,E2 -1881.995} C_VEL
LIN {X 0,Y 580.224,Z 450.435,A -85,B 0,C 180,E1 -1882.694,E2 -1882.694} C_VEL
LIN {X 0,Y 580.218,Z 458.418,A -85,B 0,C 180,E1 -1883.503,E2 -1883.503} C_VEL
LIN {X 0,Y 580.173,Z 464.436,A -85,B 0,C 180,E1 -1884.265,E2 -1884.265} C_VEL
LIN {X 0,Y 580.084,Z 469.989,A -85,B 0,C 180,E1 -1885.135,E2 -1885.135} C_VEL
LIN {X 0,Y 580.137,Z 475.15,A -85,B 0,C 180,E1 -1886.18,E2 -1886.18} C_VEL
LIN {X 0,Y 580.07,Z 477.79,A -85,B 0,C 180,E1 -1886.875,E2 -1886.875} C_VEL
LIN {X 0,Y 580.041,Z 480.682,A -85,B 0,C 180,E1 -1887.917,E2 -1887.917} C_VEL
LIN {X 0,Y 580.045,Z 481.936,A -85,B 0,C 180,E1 -1888.612,E2 -1888.612} C_VEL
LIN {X 0,Y 580.036,Z 482.711,A -85,B 0,C 180,E1 -1889.306,E2 -1889.306} C_VEL
LIN {X 0,Y 580.034,Z 483,A -85,B 0,C 180,E1 -1890,E2 -1890} C_VEL
LIN {X 0,Y 580.036,Z 482.71,A -85,B 0,C 180,E1 -1890.695,E2 -1890.695} C_VEL
LIN {X 0,Y 580.045,Z 481.935,A -85,B 0,C 180,E1 -1891.389,E2 -1891.389} C_VEL
LIN {X 0,Y 580.041,Z 480.68,A -85,B 0,C 180,E1 -1892.083,E2 -1892.083} C_VEL
LIN {X 0,Y 580.07,Z 477.787,A -85,B 0,C 180,E1 -1893.126,E2 -1893.126} C_VEL
LIN {X 0,Y 580.137,Z 475.146,A -85,B 0,C 180,E1 -1893.821,E2 -1893.821} C_VEL
LIN {X 0,Y 580.084,Z 469.984,A -85,B 0,C 180,E1 -1894.865,E2 -1894.865} C_VEL
LIN {X 0,Y 580.193,Z 463.184,A -85,B 0,C 180,E1 -1895.91,E2 -1895.91} C_VEL
LIN {X 0,Y 580.225,Z 455.493,A -85,B 0,C 180,E1 -1896.808,E2 -1896.808} C_VEL
LIN {X 0,Y 580.253,Z 448.403,A -85,B 0,C 180,E1 -1897.482,E2 -1897.482} C_VEL
LIN {X 0,Y 580.297,Z 440.542,A -85,B 0,C 180,E1 -1898.094,E2 -1898.094} C_VEL
LIN {X 0,Y 580.348,Z 430.726,A -85,B 0,C 180,E1 -1898.707,E2 -1898.707} C_VEL
LIN {X 0,Y 580.399,Z 419.293,A -85,B 0,C 180,E1 -1899.233,E2 -1899.233} C_VEL
LIN {X 0,Y 580.464,Z 409.234,A -85,B 0,C 180,E1 -1899.561,E2 -1899.561} C_VEL
LIN {X 0,Y 580.508,Z 400.424,A -85,B 0,C 180,E1 -1899.759,E2 -1899.759} C_VEL
LIN {X 0,Y 580.572,Z 331.032,A -85,B 0,C 180,E1 -1900.634,E2 -1900.634} C_VEL
LIN {X 0,Y 580.321,Z 323.3,A -85,B 0,C 180,E1 -1900.734,E2 -1900.734} C_VEL
LIN {X 0,Y 580.186,Z 322.168,A -85,B 0,C 180,E1 -1900.774,E2 -1900.774} C_VEL
LIN {X 0,Y 580.351,Z 305.23,A -85,B 0,C 180,E1 -1903.303,E2 -1903.303} C_VEL
LIN {X 0,Y 580.465,Z 286.24,A -85,B 0,C 180,E1 -1906.169,E2 -1906.169} C_VEL
LIN {X 0,Y 580.588,Z 269.625,A -85,B 0,C 180,E1 -1908.71,E2 -1908.71} C_VEL
LIN {X 0,Y 580.767,Z 251.807,A -85,B 0,C 180,E1 -1911.473,E2 -1911.473} C_VEL
LIN {X 0,Y 580.671,Z 245.685,A -85,B 0,C 180,E1 -1912.412,E2 -1912.412} C_VEL
LIN {X 0,Y 580.246,Z 243.021,A -85,B 0,C 180,E1 -1912.86,E2 -1912.86} C_VEL
LIN {X 0,Y 580.239,Z 243.019,A -85,B 0,C 180,E1 -1915.852,E2 -1915.852} C_VEL
LIN {X 0,Y 580.222,Z 243.017,A -85,B 0,C 180,E1 -1918.19,E2 -1918.19} C_VEL
LIN {X 0,Y 580.238,Z 243.016,A -85,B 0,C 180,E1 -1920.687,E2 -1920.687} C_VEL
LIN {X 0,Y 580.247,Z 243.023,A -85,B 0,C 180,E1 -1923.308,E2 -1923.308} C_VEL
LIN {X 0,Y 580.202,Z 243.022,A -85,B 0,C 180,E1 -1925.75,E2 -1925.75} C_VEL
LIN {X 0,Y 580.233,Z 243.016,A -85,B 0,C 180,E1 -1928.151,E2 -1928.151} C_VEL
LIN {X 0,Y 580.247,Z 243.019,A -85,B 0,C 180,E1 -1930.848,E2 -1930.848} C_VEL
LIN {X 0,Y 580.225,Z 243.018,A -85,B 0,C 180,E1 -1933.663,E2 -1933.663} C_VEL
LIN {X 0,Y 580.233,Z 243.017,A -85,B 0,C 180,E1 -1936.338,E2 -1936.338} C_VEL
LIN {X 0,Y 580.248,Z 243.021,A -85,B 0,C 180,E1 -1939.152,E2 -1939.152} C_VEL
LIN {X 0,Y 580.239,Z 243.015,A -85,B 0,C 180,E1 -1941.934,E2 -1941.934} C_VEL
LIN {X 0,Y 580.205,Z 243.023,A -85,B 0,C 180,E1 -1944.449,E2 -1944.449} C_VEL
LIN {X 0,Y 580.239,Z 243.022,A -85,B 0,C 180,E1 -1946.972,E2 -1946.972} C_VEL
LIN {X 0,Y 580.249,Z 243.015,A -85,B 0,C 180,E1 -1949.422,E2 -1949.422} C_VEL
LIN {X 0,Y 580.237,Z 243.018,A -85,B 0,C 180,E1 -1952.153,E2 -1952.153} C_VEL
LIN {X 0,Y 580.237,Z 243.021,A -85,B 0,C 180,E1 -1954.917,E2 -1954.917} C_VEL
LIN {X 0,Y 580.246,Z 243.016,A -85,B 0,C 180,E1 -1957.196,E2 -1957.196} C_VEL
LIN {X 0,Y 580.24,Z 243.015,A -85,B 0,C 180,E1 -1959.436,E2 -1959.436} C_VEL
LIN {X 0,Y 580.234,Z 243.024,A -85,B 0,C 180,E1 -1962.374,E2 -1962.374} C_VEL
LIN {X 0,Y 580.259,Z 243.013,A -85,B 0,C 180,E1 -1965.265,E2 -1965.265} C_VEL
LIN {X 0,Y 580.281,Z 243.016,A -85,B 0,C 180,E1 -1968.118,E2 -1968.118} C_VEL
LIN {X 0,Y 580.235,Z 243.017,A -85,B 0,C 180,E1 -1970.941,E2 -1970.941} C_VEL
LIN {X 0,Y 580.256,Z 243.016,A -85,B 0,C 180,E1 -1973.742,E2 -1973.742} C_VEL
LIN {X 0,Y 580.252,Z 243.018,A -85,B 0,C 180,E1 -1975.833,E2 -1975.833} C_VEL
LIN {X 0,Y 580.337,Z 243.009,A -85,B 0,C 180,E1 -1977.918,E2 -1977.918} C_VEL
LIN {X 0,Y 580.348,Z 243.01,A -85,B 0,C 180,E1 -1980,E2 -1980} C_VEL
LIN {X 0,Y 580.302,Z 243.008,A -85,B 0,C 180,E1 -1982.777,E2 -1982.777} C_VEL
LIN {X 0,Y 580.296,Z 243.011,A -85,B 0,C 180,E1 -1985.56,E2 -1985.56} C_VEL
LIN {X 0,Y 580.293,Z 243.012,A -85,B 0,C 180,E1 -1988.357,E2 -1988.357} C_VEL
LIN {X 0,Y 580.269,Z 243.013,A -85,B 0,C 180,E1 -1991.174,E2 -1991.174} C_VEL
LIN {X 0,Y 580.294,Z 243.016,A -85,B 0,C 180,E1 -1994.018,E2 -1994.018} C_VEL
LIN {X 0,Y 580.251,Z 243.014,A -85,B 0,C 180,E1 -1996.899,E2 -1996.899} C_VEL
LIN {X 0,Y 580.269,Z 243.02,A -85,B 0,C 180,E1 -1999.824,E2 -1999.824} C_VEL
LIN {X 0,Y 580.265,Z 243.016,A -85,B 0,C 180,E1 -2001.287,E2 -2001.287} C_VEL
LIN {X 0,Y 579.614,Z 243.103,A -85,B 0,C 180,E1 -2001.866,E2 -2001.866} C_VEL
LIN {X 0,Y 576.735,Z 243.462,A -85,B 0,C 180,E1 -2002.806,E2 -2002.806} C_VEL
LIN {X 0,Y 574.3,Z 243.764,A -85,B 0,C 180,E1 -2003.562,E2 -2003.562} C_VEL
LIN {X 0,Y 573.269,Z 243.886,A -85,B 0,C 180,E1 -2004.146,E2 -2004.146} C_VEL
LIN {X 0,Y 573.194,Z 243.894,A -85,B 0,C 180,E1 -2004.344,E2 -2004.344} C_VEL
LIN {X 0,Y 573.188,Z 243.896,A -85,B 0,C 180,E1 -2006.979,E2 -2006.979} C_VEL
LIN {X 0,Y 573.2,Z 243.901,A -85,B 0,C 180,E1 -2009.479,E2 -2009.479} C_VEL
LIN {X 0,Y 573.236,Z 243.888,A -85,B 0,C 180,E1 -2012.225,E2 -2012.225} C_VEL
LIN {X 0,Y 573.219,Z 243.891,A -85,B 0,C 180,E1 -2014.769,E2 -2014.769} C_VEL
LIN {X 0,Y 573.221,Z 243.893,A -85,B 0,C 180,E1 -2017.809,E2 -2017.809} C_VEL
LIN {X 0,Y 573.229,Z 243.889,A -85,B 0,C 180,E1 -2020.527,E2 -2020.527} C_VEL
LIN {X 0,Y 573.206,Z 243.895,A -85,B 0,C 180,E1 -2023.665,E2 -2023.665} C_VEL
LIN {X 0,Y 573.2,Z 243.895,A -85,B 0,C 180,E1 -2026.637,E2 -2026.637} C_VEL
LIN {X 0,Y 573.247,Z 243.891,A -85,B 0,C 180,E1 -2029.475,E2 -2029.475} C_VEL
LIN {X 0,Y 573.226,Z 243.889,A -85,B 0,C 180,E1 -2032.191,E2 -2032.191} C_VEL
LIN {X 0,Y 573.221,Z 243.896,A -85,B 0,C 180,E1 -2035.231,E2 -2035.231} C_VEL
LIN {X 0,Y 573.237,Z 243.888,A -85,B 0,C 180,E1 -2037.774,E2 -2037.774} C_VEL
LIN {X 0,Y 573.232,Z 243.894,A -85,B 0,C 180,E1 -2040.632,E2 -2040.632} C_VEL
LIN {X 0,Y 573.21,Z 243.892,A -85,B 0,C 180,E1 -2043.513,E2 -2043.513} C_VEL
LIN {X 0,Y 573.195,Z 243.894,A -85,B 0,C 180,E1 -2046.133,E2 -2046.133} C_VEL
LIN {X 0,Y 573.228,Z 243.892,A -85,B 0,C 180,E1 -2049.172,E2 -2049.172} C_VEL
LIN {X 0,Y 573.196,Z 243.893,A -85,B 0,C 180,E1 -2051.41,E2 -2051.41} C_VEL
LIN {X 0,Y 573.23,Z 243.896,A -85,B 0,C 180,E1 -2054.169,E2 -2054.169} C_VEL
LIN {X 0,Y 573.089,Z 256.901,A -85,B 0,C 180,E1 -2057.247,E2 -2057.247} C_VEL
LIN {X 0,Y 573.021,Z 265.171,A -85,B 0,C 180,E1 -2059.186,E2 -2059.186} C_VEL
LIN {X 0,Y 573.636,Z 270.396,A -85,B 0,C 180,E1 -2059.273,E2 -2059.273} C_VEL
LIN {X 0,Y 573.512,Z 340.391,A -85,B 0,C 180,E1 -2060.166,E2 -2060.166} C_VEL
LIN {X 0,Y 573.441,Z 350.046,A -85,B 0,C 180,E1 -2060.387,E2 -2060.387} C_VEL
LIN {X 0,Y 573.367,Z 361.593,A -85,B 0,C 180,E1 -2060.786,E2 -2060.786} C_VEL
LIN {X 0,Y 573.332,Z 371.463,A -85,B 0,C 180,E1 -2061.275,E2 -2061.275} C_VEL
LIN {X 0,Y 573.272,Z 379.913,A -85,B 0,C 180,E1 -2061.806,E2 -2061.806} C_VEL
LIN {X 0,Y 573.217,Z 387.882,A -85,B 0,C 180,E1 -2062.426,E2 -2062.426} C_VEL
LIN {X 0,Y 573.164,Z 393.606,A -85,B 0,C 180,E1 -2062.956,E2 -2062.956} C_VEL
LIN {X 0,Y 573.129,Z 399.995,A -85,B 0,C 180,E1 -2063.663,E2 -2063.663} C_VEL
LIN {X 0,Y 573.051,Z 406.48,A -85,B 0,C 180,E1 -2064.546,E2 -2064.546} C_VEL
LIN {X 0,Y 573.039,Z 411.653,A -85,B 0,C 180,E1 -2065.427,E2 -2065.427} C_VEL
LIN {X 0,Y 573.025,Z 416.45,A -85,B 0,C 180,E1 -2066.484,E2 -2066.484} C_VEL
LIN {X 0,Y 572.962,Z 418.787,A -85,B 0,C 180,E1 -2067.187,E2 -2067.187} C_VEL
LIN {X 0,Y 572.941,Z 420.578,A -85,B 0,C 180,E1 -2067.891,E2 -2067.891} C_VEL
LIN {X 0,Y 572.944,Z 421.871,A -85,B 0,C 180,E1 -2068.594,E2 -2068.594} C_VEL
LIN {X 0,Y 572.936,Z 422.688,A -85,B 0,C 180,E1 -2069.297,E2 -2069.297} C_VEL
LIN {X 0,Y 572.936,Z 422.996,A -85,B 0,C 180,E1 -2070,E2 -2070} C_VEL
LIN {X 0,Y 572.937,Z 422.73,A -85,B 0,C 180,E1 -2070.702,E2 -2070.702} C_VEL
LIN {X 0,Y 572.945,Z 421.996,A -85,B 0,C 180,E1 -2071.405,E2 -2071.405} C_VEL
LIN {X 0,Y 572.941,Z 420.785,A -85,B 0,C 180,E1 -2072.109,E2 -2072.109} C_VEL
LIN {X 0,Y 572.991,Z 417.937,A -85,B 0,C 180,E1 -2073.164,E2 -2073.164} C_VEL
LIN {X 0,Y 573.025,Z 415.344,A -85,B 0,C 180,E1 -2073.867,E2 -2073.867} C_VEL
LIN {X 0,Y 572.983,Z 410.235,A -85,B 0,C 180,E1 -2074.925,E2 -2074.925} C_VEL
LIN {X 0,Y 573.113,Z 404.737,A -85,B 0,C 180,E1 -2075.806,E2 -2075.806} C_VEL
LIN {X 0,Y 573.156,Z 396.341,A -85,B 0,C 180,E1 -2076.849,E2 -2076.849} C_VEL
LIN {X 0,Y 573.215,Z 388.923,A -85,B 0,C 180,E1 -2077.573,E2 -2077.573} C_VEL
LIN {X 0,Y 573.302,Z 381.169,A -85,B 0,C 180,E1 -2078.193,E2 -2078.193} C_VEL
LIN {X 0,Y 573.337,Z 372.995,A -85,B 0,C 180,E1 -2078.725,E2 -2078.725} C_VEL
LIN {X 0,Y 573.373,Z 362.606,A -85,B 0,C 180,E1 -2079.257,E2 -2079.257} C_VEL
LIN {X 0,Y 573.422,Z 350.937,A -85,B 0,C 180,E1 -2079.679,E2 -2079.679} C_VEL
LIN {X 0,Y 573.536,Z 340.491,A -85,B 0,C 180,E1 -2079.922,E2 -2079.922} C_VEL
LIN {X 0,Y 573.607,Z 292.193,A -85,B 0,C 180,E1 -2080.545,E2 -2080.545} C_VEL
LIN {X 0,Y 573.442,Z 268.323,A -85,B 0,C 180,E1 -2080.846,E2 -2080.846} C_VEL
LIN {X 0,Y 573.048,Z 265.095,A -85,B 0,C 180,E1 -2080.922,E2 -2080.922} C_VEL
LIN {X 0,Y 573.135,Z 252.695,A -85,B 0,C 180,E1 -2083.834,E2 -2083.834} C_VEL
LIN {X 0,Y 573.211,Z 243.896,A -85,B 0,C 180,E1 -2085.922,E2 -2085.922} C_VEL
LIN {X 0,Y 573.269,Z 243.891,A -85,B 0,C 180,E1 -2089.268,E2 -2089.268} C_VEL
LIN {X 0,Y 573.194,Z 243.893,A -85,B 0,C 180,E1 -2092.339,E2 -2092.339} C_VEL
LIN {X 0,Y 573.221,Z 243.898,A -85,B 0,C 180,E1 -2095.411,E2 -2095.411} C_VEL
LIN {X 0,Y 573.193,Z 243.894,A -85,B 0,C 180,E1 -2098.018,E2 -2098.018} C_VEL
LIN {X 0,Y 573.208,Z 243.896,A -85,B 0,C 180,E1 -2100.878,E2 -2100.878} C_VEL
LIN {X 0,Y 573.239,Z 243.891,A -85,B 0,C 180,E1 -2103.52,E2 -2103.52} C_VEL
LIN {X 0,Y 573.179,Z 243.895,A -85,B 0,C 180,E1 -2106.053,E2 -2106.053} C_VEL
LIN {X 0,Y 573.228,Z 243.894,A -85,B 0,C 180,E1 -2108.702,E2 -2108.702} C_VEL
LIN {X 0,Y 573.196,Z 243.895,A -85,B 0,C 180,E1 -2111.459,E2 -2111.459} C_VEL
LIN {X 0,Y 573.213,Z 243.893,A -85,B 0,C 180,E1 -2114.335,E2 -2114.335} C_VEL
LIN {X 0,Y 573.209,Z 243.894,A -85,B 0,C 180,E1 -2117.361,E2 -2117.361} C_VEL
LIN {X 0,Y 573.223,Z 243.894,A -85,B 0,C 180,E1 -2120.391,E2 -2120.391} C_VEL
LIN {X 0,Y 573.224,Z 243.894,A -85,B 0,C 180,E1 -2123.075,E2 -2123.075} C_VEL
LIN {X 0,Y 573.237,Z 243.888,A -85,B 0,C 180,E1 -2125.669,E2 -2125.669} C_VEL
LIN {X 0,Y 573.219,Z 243.894,A -85,B 0,C 180,E1 -2128.183,E2 -2128.183} C_VEL
LIN {X 0,Y 573.21,Z 243.9,A -85,B 0,C 180,E1 -2130.631,E2 -2130.631} C_VEL
LIN {X 0,Y 573.198,Z 243.893,A -85,B 0,C 180,E1 -2133.514,E2 -2133.514} C_VEL
LIN {X 0,Y 573.187,Z 243.899,A -85,B 0,C 180,E1 -2136.132,E2 -2136.132} C_VEL
LIN {X 0,Y 573.22,Z 243.89,A -85,B 0,C 180,E1 -2139.172,E2 -2139.172} C_VEL
LIN {X 0,Y 573.186,Z 243.894,A -85,B 0,C 180,E1 -2141.41,E2 -2141.41} C_VEL
LIN {X 0,Y 573.196,Z 243.901,A -85,B 0,C 180,E1 -2144.351,E2 -2144.351} C_VEL
LIN {X 0,Y 573.188,Z 243.899,A -85,B 0,C 180,E1 -2146.528,E2 -2146.528} C_VEL
LIN {X 0,Y 573.235,Z 243.889,A -85,B 0,C 180,E1 -2149.403,E2 -2149.403} C_VEL
LIN {X 0,Y 573.213,Z 243.898,A -85,B 0,C 180,E1 -2152.249,E2 -2152.249} C_VEL
LIN {X 0,Y 573.268,Z 243.884,A -85,B 0,C 180,E1 -2155.077,E2 -2155.077} C_VEL
LIN {X 0,Y 573.305,Z 243.888,A -85,B 0,C 180,E1 -2157.892,E2 -2157.892} C_VEL
LIN {X 0,Y 573.311,Z 243.887,A -85,B 0,C 180,E1 -2160,E2 -2160} C_VEL
LIN {X 0,Y 573.263,Z 243.885,A -85,B 0,C 180,E1 -2162.811,E2 -2162.811} C_VEL
LIN {X 0,Y 573.263,Z 243.891,A -85,B 0,C 180,E1 -2165.628,E2 -2165.628} C_VEL
LIN {X 0,Y 573.227,Z 243.89,A -85,B 0,C 180,E1 -2168.46,E2 -2168.46} C_VEL
LIN {X 0,Y 573.229,Z 243.893,A -85,B 0,C 180,E1 -2171.313,E2 -2171.313} C_VEL
LIN {X 0,Y 573.229,Z 243.889,A -85,B 0,C 180,E1 -2174.406,E2 -2174.406} C_VEL
LIN {X 0,Y 573.185,Z 243.897,A -85,B 0,C 180,E1 -2177.114,E2 -2177.114} C_VEL
LIN {X 0,Y 573.196,Z 243.895,A -85,B 0,C 180,E1 -2180.079,E2 -2180.079} C_VEL
LIN {X 0,Y 573.188,Z 243.894,A -85,B 0,C 180,E1 -2182.34,E2 -2182.34} C_VEL
LIN {X 0,Y 573.203,Z 243.901,A -85,B 0,C 180,E1 -2185.412,E2 -2185.412} C_VEL
LIN {X 0,Y 573.187,Z 243.895,A -85,B 0,C 180,E1 -2188.018,E2 -2188.018} C_VEL
LIN {X 0,Y 573.197,Z 243.896,A -85,B 0,C 180,E1 -2190.878,E2 -2190.878} C_VEL
LIN {X 0,Y 573.236,Z 243.893,A -85,B 0,C 180,E1 -2193.521,E2 -2193.521} C_VEL
LIN {X 0,Y 573.175,Z 243.895,A -85,B 0,C 180,E1 -2196.054,E2 -2196.054} C_VEL
LIN {X 0,Y 573.221,Z 243.893,A -85,B 0,C 180,E1 -2198.703,E2 -2198.703} C_VEL
LIN {X 0,Y 573.189,Z 243.896,A -85,B 0,C 180,E1 -2201.589,E2 -2201.589} C_VEL
LIN {X 0,Y 573.202,Z 243.897,A -85,B 0,C 180,E1 -2204.674,E2 -2204.674} C_VEL
LIN {X 0,Y 573.198,Z 243.893,A -85,B 0,C 180,E1 -2207.597,E2 -2207.597} C_VEL
LIN {X 0,Y 573.225,Z 243.894,A -85,B 0,C 180,E1 -2210.571,E2 -2210.571} C_VEL
LIN {X 0,Y 573.22,Z 243.895,A -85,B 0,C 180,E1 -2213.076,E2 -2213.076} C_VEL
LIN {X 0,Y 573.229,Z 243.888,A -85,B 0,C 180,E1 -2215.669,E2 -2215.669} C_VEL
LIN {X 0,Y 573.202,Z 243.894,A -85,B 0,C 180,E1 -2218.183,E2 -2218.183} C_VEL
LIN {X 0,Y 573.209,Z 243.9,A -85,B 0,C 180,E1 -2220.632,E2 -2220.632} C_VEL
LIN {X 0,Y 573.188,Z 243.894,A -85,B 0,C 180,E1 -2223.517,E2 -2223.517} C_VEL
LIN {X 0,Y 573.184,Z 243.899,A -85,B 0,C 180,E1 -2226.133,E2 -2226.133} C_VEL
LIN {X 0,Y 573.231,Z 244.053,A -85,B 0,C 180,E1 -2227.092,E2 -2227.092} C_VEL
LIN {X 0,Y 573.805,Z 248.977,A -85,B 0,C 180,E1 -2227.876,E2 -2227.876} C_VEL
LIN {X 0,Y 573.661,Z 266.843,A -85,B 0,C 180,E1 -2230.62,E2 -2230.62} C_VEL
LIN {X 0,Y 573.52,Z 283.982,A -85,B 0,C 180,E1 -2233.281,E2 -2233.281} C_VEL
LIN {X 0,Y 573.375,Z 302.861,A -85,B 0,C 180,E1 -2236.172,E2 -2236.172} C_VEL
LIN {X 0,Y 573.162,Z 322.065,A -85,B 0,C 180,E1 -2239.077,E2 -2239.077} C_VEL
LIN {X 0,Y 573.198,Z 322.896,A -85,B 0,C 180,E1 -2239.126,E2 -2239.126} C_VEL
LIN {X 0,Y 573.622,Z 328.424,A -85,B 0,C 180,E1 -2239.203,E2 -2239.203} C_VEL
LIN {X 0,Y 573.552,Z 399.163,A -85,B 0,C 180,E1 -2240.1,E2 -2240.1} C_VEL
LIN {X 0,Y 573.453,Z 408.428,A -85,B 0,C 180,E1 -2240.299,E2 -2240.299} C_VEL
LIN {X 0,Y 573.42,Z 416.901,A -85,B 0,C 180,E1 -2240.565,E2 -2240.565} C_VEL
LIN {X 0,Y 573.349,Z 425.406,A -85,B 0,C 180,E1 -2240.92,E2 -2240.92} C_VEL
LIN {X 0,Y 573.332,Z 433.736,A -85,B 0,C 180,E1 -2241.364,E2 -2241.364} C_VEL
